LIN {X 0,Y 475.788,Z 378.361,A -85,B 0,C 180,E1 -7451.438,E2 -7451.438} C_VEL
LIN {X 0,Y 475.279,Z 381.668,A -85,B 0,C 180,E1 -7452.005,E2 -7452.005} C_VEL
LIN {X 0,Y 474.286,Z 385.768,A -85,B 0,C 180,E1 -7452.486,E2 -7452.486} C_VEL
LIN {X 0,Y 473.126,Z 390.462,A -85,B 0,C 180,E1 -7452.878,E2 -7452.878} C_VEL
LIN {X 0,Y 471.802,Z 397.453,A -85,B 0,C 180,E1 -7453.254,E2 -7453.254} C_VEL
LIN {X 0,Y 471.382,Z 403.104,A -85,B 0,C 180,E1 -7453.407,E2 -7453.407} C_VEL
LIN {X 0,Y 470.706,Z 494.322,A -85,B 0,C 180,E1 -7454.826,E2 -7454.826} C_VEL
LIN {X 0,Y 470.353,Z 508.19,A -85,B 0,C 180,E1 -7455.23,E2 -7455.23} C_VEL
LIN {X 0,Y 470.018,Z 520.592,A -85,B 0,C 180,E1 -7455.772,E2 -7455.772} C_VEL
LIN {X 0,Y 469.61,Z 532.37,A -85,B 0,C 180,E1 -7456.472,E2 -7456.472} C_VEL
LIN {X 0,Y 469.141,Z 543.794,A -85,B 0,C 180,E1 -7457.345,E2 -7457.345} C_VEL
LIN {X 0,Y 468.592,Z 554.026,A -85,B 0,C 180,E1 -7458.319,E2 -7458.319} C_VEL
LIN {X 0,Y 468.161,Z 563.202,A -85,B 0,C 180,E1 -7459.403,E2 -7459.403} C_VEL
LIN {X 0,Y 467.689,Z 572.108,A -85,B 0,C 180,E1 -7460.704,E2 -7460.704} C_VEL
LIN {X 0,Y 467.314,Z 579.277,A -85,B 0,C 180,E1 -7462.004,E2 -7462.004} C_VEL
LIN {X 0,Y 467.081,Z 584.816,A -85,B 0,C 180,E1 -7463.257,E2 -7463.257} C_VEL
LIN {X 0,Y 466.93,Z 588.808,A -85,B 0,C 180,E1 -7464.386,E2 -7464.386} C_VEL
LIN {X 0,Y 466.822,Z 592.404,A -85,B 0,C 180,E1 -7465.683,E2 -7465.683} C_VEL
LIN {X 0,Y 466.78,Z 594.262,A -85,B 0,C 180,E1 -7466.547,E2 -7466.547} C_VEL
LIN {X 0,Y 466.704,Z 595.664,A -85,B 0,C 180,E1 -7467.411,E2 -7467.411} C_VEL
LIN {X 0,Y 466.62,Z 597.275,A -85,B 0,C 180,E1 -7469.137,E2 -7469.137} C_VEL
LIN {X 0,Y 466.6,Z 597.511,A -85,B 0,C 180,E1 -7470,E2 -7470} C_VEL
LIN {X 0,Y 466.62,Z 597.325,A -85,B 0,C 180,E1 -7470.863,E2 -7470.863} C_VEL
LIN {X 0,Y 466.704,Z 595.778,A -85,B 0,C 180,E1 -7472.589,E2 -7472.589} C_VEL
LIN {X 0,Y 466.78,Z 594.425,A -85,B 0,C 180,E1 -7473.453,E2 -7473.453} C_VEL
LIN {X 0,Y 466.788,Z 591.571,A -85,B 0,C 180,E1 -7474.75,E2 -7474.75} C_VEL
LIN {X 0,Y 467.034,Z 587.692,A -85,B 0,C 180,E1 -7476.046,E2 -7476.046} C_VEL
LIN {X 0,Y 467.17,Z 582.693,A -85,B 0,C 180,E1 -7477.346,E2 -7477.346} C_VEL
LIN {X 0,Y 467.441,Z 576.398,A -85,B 0,C 180,E1 -7478.647,E2 -7478.647} C_VEL
LIN {X 0,Y 467.856,Z 568.513,A -85,B 0,C 180,E1 -7479.947,E2 -7479.947} C_VEL
LIN {X 0,Y 468.293,Z 558.704,A -85,B 0,C 180,E1 -7481.25,E2 -7481.25} C_VEL
LIN {X 0,Y 468.93,Z 548.404,A -85,B 0,C 180,E1 -7482.331,E2 -7482.331} C_VEL
LIN {X 0,Y 469.328,Z 537.488,A -85,B 0,C 180,E1 -7483.256,E2 -7483.256} C_VEL
LIN {X 0,Y 469.796,Z 527.044,A -85,B 0,C 180,E1 -7483.959,E2 -7483.959} C_VEL
LIN {X 0,Y 470.212,Z 514.491,A -85,B 0,C 180,E1 -7484.609,E2 -7484.609} C_VEL
LIN {X 0,Y 470.562,Z 501.002,A -85,B 0,C 180,E1 -7485.095,E2 -7485.095} C_VEL
LIN {X 0,Y 470.722,Z 487.471,A -85,B 0,C 180,E1 -7485.395,E2 -7485.395} C_VEL
LIN {X 0,Y 471.408,Z 402.034,A -85,B 0,C 180,E1 -7486.7,E2 -7486.7} C_VEL
LIN {X 0,Y 468.486,Z 387.239,A -85,B 0,C 180,E1 -7487.057,E2 -7487.057} C_VEL
LIN {X 0,Y 468.974,Z 376.155,A -85,B 0,C 180,E1 -7489.477,E2 -7489.477} C_VEL
LIN {X 0,Y 467.573,Z 368.247,A -85,B 0,C 180,E1 -7491.388,E2 -7491.388} C_VEL
LIN {X 0,Y 467.575,Z 368.247,A -85,B 0,C 180,E1 -7493.943,E2 -7493.943} C_VEL
LIN {X 0,Y 467.617,Z 368.232,A -85,B 0,C 180,E1 -7496.8,E2 -7496.8} C_VEL
LIN {X 0,Y 467.554,Z 368.245,A -85,B 0,C 180,E1 -7499.737,E2 -7499.737} C_VEL
LIN {X 0,Y 467.583,Z 368.236,A -85,B 0,C 180,E1 -7502.758,E2 -7502.758} C_VEL
LIN {X 0,Y 467.555,Z 368.248,A -85,B 0,C 180,E1 -7505.888,E2 -7505.888} C_VEL
LIN {X 0,Y 467.58,Z 368.237,A -85,B 0,C 180,E1 -7509.144,E2 -7509.144} C_VEL
LIN {X 0,Y 467.583,Z 368.236,A -85,B 0,C 180,E1 -7512.566,E2 -7512.566} C_VEL
LIN {X 0,Y 467.567,Z 368.239,A -85,B 0,C 180,E1 -7515.052,E2 -7515.052} C_VEL
LIN {X 0,Y 467.62,Z 368.236,A -85,B 0,C 180,E1 -7517.443,E2 -7517.443} C_VEL
LIN {X 0,Y 467.595,Z 368.235,A -85,B 0,C 180,E1 -7520.856,E2 -7520.856} C_VEL
LIN {X 0,Y 467.558,Z 368.24,A -85,B 0,C 180,E1 -7524.26,E2 -7524.26} C_VEL
LIN {X 0,Y 467.583,Z 368.241,A -85,B 0,C 180,E1 -7527.319,E2 -7527.319} C_VEL
LIN {X 0,Y 467.563,Z 368.239,A -85,B 0,C 180,E1 -7530.667,E2 -7530.667} C_VEL
LIN {X 0,Y 467.621,Z 368.236,A -85,B 0,C 180,E1 -7533.2,E2 -7533.2} C_VEL
LIN {X 0,Y 467.586,Z 368.236,A -85,B 0,C 180,E1 -7536.467,E2 -7536.467} C_VEL
LIN {X 0,Y 467.616,Z 368.235,A -85,B 0,C 180,E1 -7539.777,E2 -7539.777} C_VEL
LIN {X 0,Y 467.601,Z 368.234,A -85,B 0,C 180,E1 -7542.506,E2 -7542.506} C_VEL
LIN {X 0,Y 467.601,Z 368.241,A -85,B 0,C 180,E1 -7545.196,E2 -7545.196} C_VEL
LIN {X 0,Y 467.674,Z 368.226,A -85,B 0,C 180,E1 -7547.855,E2 -7547.855} C_VEL
LIN {X 0,Y 467.674,Z 368.231,A -85,B 0,C 180,E1 -7551.357,E2 -7551.357} C_VEL
LIN {X 0,Y 467.735,Z 368.218,A -85,B 0,C 180,E1 -7553.962,E2 -7553.962} C_VEL
LIN {X 0,Y 467.853,Z 368.207,A -85,B 0,C 180,E1 -7557.417,E2 -7557.417} C_VEL
LIN {X 0,Y 467.873,Z 368.2,A -85,B 0,C 180,E1 -7560,E2 -7560} C_VEL
LIN {X 0,Y 467.853,Z 368.205,A -85,B 0,C 180,E1 -7562.583,E2 -7562.583} C_VEL
LIN {X 0,Y 467.739,Z 368.217,A -85,B 0,C 180,E1 -7566.037,E2 -7566.037} C_VEL
LIN {X 0,Y 467.674,Z 368.228,A -85,B 0,C 180,E1 -7568.643,E2 -7568.643} C_VEL
LIN {X 0,Y 467.674,Z 368.225,A -85,B 0,C 180,E1 -7572.145,E2 -7572.145} C_VEL
LIN {X 0,Y 467.641,Z 368.229,A -85,B 0,C 180,E1 -7575.886,E2 -7575.886} C_VEL
LIN {X 0,Y 467.616,Z 368.234,A -85,B 0,C 180,E1 -7579.308,E2 -7579.308} C_VEL
LIN {X 0,Y 467.534,Z 368.243,A -85,B 0,C 180,E1 -7582.074,E2 -7582.074} C_VEL
LIN {X 0,Y 467.598,Z 368.241,A -85,B 0,C 180,E1 -7584.888,E2 -7584.888} C_VEL
LIN {X 0,Y 467.62,Z 368.232,A -85,B 0,C 180,E1 -7587.769,E2 -7587.769} C_VEL
LIN {X 0,Y 467.562,Z 368.242,A -85,B 0,C 180,E1 -7591.046,E2 -7591.046} C_VEL
LIN {X 0,Y 467.584,Z 368.239,A -85,B 0,C 180,E1 -7594.243,E2 -7594.243} C_VEL
LIN {X 0,Y 467.545,Z 368.242,A -85,B 0,C 180,E1 -7597.188,E2 -7597.188} C_VEL
LIN {X 0,Y 467.591,Z 368.24,A -85,B 0,C 180,E1 -7600.263,E2 -7600.263} C_VEL
LIN {X 0,Y 467.615,Z 368.24,A -85,B 0,C 180,E1 -7602.572,E2 -7602.572} C_VEL
LIN {X 0,Y 467.563,Z 368.243,A -85,B 0,C 180,E1 -7606.178,E2 -7606.178} C_VEL
LIN {X 0,Y 467.579,Z 368.241,A -85,B 0,C 180,E1 -7608.723,E2 -7608.723} C_VEL
LIN {X 0,Y 467.564,Z 368.242,A -85,B 0,C 180,E1 -7611.956,E2 -7611.956} C_VEL
LIN {X 0,Y 467.567,Z 368.238,A -85,B 0,C 180,E1 -7615.169,E2 -7615.169} C_VEL
LIN {X 0,Y 467.583,Z 368.244,A -85,B 0,C 180,E1 -7618.261,E2 -7618.261} C_VEL
LIN {X 0,Y 467.576,Z 368.241,A -85,B 0,C 180,E1 -7621.251,E2 -7621.251} C_VEL
LIN {X 0,Y 467.669,Z 368.367,A -85,B 0,C 180,E1 -7623.805,E2 -7623.805} C_VEL
LIN {X 0,Y 469.783,Z 379.089,A -85,B 0,C 180,E1 -7625.863,E2 -7625.863} C_VEL
LIN {X 0,Y 469.854,Z 384.768,A -85,B 0,C 180,E1 -7626.882,E2 -7626.882} C_VEL
LIN {X 0,Y 469.109,Z 400.416,A -85,B 0,C 180,E1 -7629.616,E2 -7629.616} C_VEL
LIN {X 0,Y 468.442,Z 417.254,A -85,B 0,C 180,E1 -7632.539,E2 -7632.539} C_VEL
LIN {X 0,Y 468.328,Z 419.783,A -85,B 0,C 180,E1 -7632.978,E2 -7632.978} C_VEL
LIN {X 0,Y 471.197,Z 439.463,A -85,B 0,C 180,E1 -7633.391,E2 -7633.391} C_VEL
LIN {X 0,Y 470.547,Z 528.128,A -85,B 0,C 180,E1 -7634.765,E2 -7634.765} C_VEL
LIN {X 0,Y 470.162,Z 541.402,A -85,B 0,C 180,E1 -7635.141,E2 -7635.141} C_VEL
LIN {X 0,Y 469.689,Z 554.694,A -85,B 0,C 180,E1 -7635.707,E2 -7635.707} C_VEL
LIN {X 0,Y 469.247,Z 565.855,A -85,B 0,C 180,E1 -7636.356,E2 -7636.356} C_VEL
LIN {X 0,Y 468.69,Z 577.047,A -85,B 0,C 180,E1 -7637.187,E2 -7637.187} C_VEL
LIN {X 0,Y 468.235,Z 587.923,A -85,B 0,C 180,E1 -7638.2,E2 -7638.2} C_VEL
LIN {X 0,Y 467.784,Z 596.474,A -85,B 0,C 180,E1 -7639.176,E2 -7639.176} C_VEL
LIN {X 0,Y 467.434,Z 604.368,A -85,B 0,C 180,E1 -7640.262,E2 -7640.262} C_VEL
LIN {X 0,Y 467.113,Z 612.079,A -85,B 0,C 180,E1 -7641.565,E2 -7641.565} C_VEL
LIN {X 0,Y 466.858,Z 619.19,A -85,B 0,C 180,E1 -7643.083,E2 -7643.083} C_VEL
LIN {X 0,Y 466.763,Z 623.924,A -85,B 0,C 180,E1 -7644.384,E2 -7644.384} C_VEL
LIN {X 0,Y 466.648,Z 627.539,A -85,B 0,C 180,E1 -7645.681,E2 -7645.681} C_VEL
LIN {X 0,Y 466.69,Z 629.407,A -85,B 0,C 180,E1 -7646.547,E2 -7646.547} C_VEL
LIN {X 0,Y 466.662,Z 630.806,A -85,B 0,C 180,E1 -7647.411,E2 -7647.411} C_VEL
LIN {X 0,Y 466.619,Z 632.413,A -85,B 0,C 180,E1 -7649.137,E2 -7649.137} C_VEL
LIN {X 0,Y 466.599,Z 632.629,A -85,B 0,C 180,E1 -7650,E2 -7650} C_VEL
LIN {X 0,Y 466.619,Z 632.413,A -85,B 0,C 180,E1 -7650.863,E2 -7650.863} C_VEL
LIN {X 0,Y 466.662,Z 630.809,A -85,B 0,C 180,E1 -7652.589,E2 -7652.589} C_VEL
LIN {X 0,Y 466.69,Z 629.41,A -85,B 0,C 180,E1 -7653.453,E2 -7653.453} C_VEL
LIN {X 0,Y 466.69,Z 626.466,A -85,B 0,C 180,E1 -7654.751,E2 -7654.751} C_VEL
LIN {X 0,Y 466.753,Z 622.483,A -85,B 0,C 180,E1 -7656.05,E2 -7656.05} C_VEL
LIN {X 0,Y 466.943,Z 616.362,A -85,B 0,C 180,E1 -7657.567,E2 -7657.567} C_VEL
LIN {X 0,Y 467.188,Z 609.672,A -85,B 0,C 180,E1 -7658.87,E2 -7658.87} C_VEL
LIN {X 0,Y 467.521,Z 601.374,A -85,B 0,C 180,E1 -7660.173,E2 -7660.173} C_VEL
LIN {X 0,Y 468.007,Z 592.876,A -85,B 0,C 180,E1 -7661.257,E2 -7661.257} C_VEL
LIN {X 0,Y 468.474,Z 582.834,A -85,B 0,C 180,E1 -7662.301,E2 -7662.301} C_VEL
LIN {X 0,Y 468.938,Z 571.987,A -85,B 0,C 180,E1 -7663.212,E2 -7663.212} C_VEL
LIN {X 0,Y 469.449,Z 560.604,A -85,B 0,C 180,E1 -7663.969,E2 -7663.969} C_VEL
LIN {X 0,Y 469.913,Z 548.932,A -85,B 0,C 180,E1 -7664.563,E2 -7664.563} C_VEL
LIN {X 0,Y 470.33,Z 536.401,A -85,B 0,C 180,E1 -7665.02,E2 -7665.02} C_VEL
LIN {X 0,Y 470.645,Z 523.722,A -85,B 0,C 180,E1 -7665.314,E2 -7665.314} C_VEL
LIN {X 0,Y 471.1,Z 437.824,A -85,B 0,C 180,E1 -7666.636,E2 -7666.636} C_VEL
LIN {X 0,Y 468.331,Z 419.732,A -85,B 0,C 180,E1 -7667.032,E2 -7667.032} C_VEL
LIN {X 0,Y 469.063,Z 401.69,A -85,B 0,C 180,E1 -7670.158,E2 -7670.158} C_VEL
LIN {X 0,Y 469.826,Z 386.056,A -85,B 0,C 180,E1 -7672.887,E2 -7672.887} C_VEL
LIN {X 0,Y 469.981,Z 380.833,A -85,B 0,C 180,E1 -7673.812,E2 -7673.812} C_VEL
LIN {X 0,Y 468.071,Z 370.311,A -85,B 0,C 180,E1 -7675.812,E2 -7675.812} C_VEL
LIN {X 0,Y 467.645,Z 368.234,A -85,B 0,C 180,E1 -7676.257,E2 -7676.257} C_VEL
LIN {X 0,Y 467.57,Z 368.244,A -85,B 0,C 180,E1 -7679.332,E2 -7679.332} C_VEL
LIN {X 0,Y 467.581,Z 368.236,A -85,B 0,C 180,E1 -7682.679,E2 -7682.679} C_VEL
LIN {X 0,Y 467.561,Z 368.246,A -85,B 0,C 180,E1 -7685.739,E2 -7685.739} C_VEL
LIN {X 0,Y 467.58,Z 368.239,A -85,B 0,C 180,E1 -7689.144,E2 -7689.144} C_VEL
LIN {X 0,Y 467.583,Z 368.236,A -85,B 0,C 180,E1 -7692.566,E2 -7692.566} C_VEL
LIN {X 0,Y 467.567,Z 368.24,A -85,B 0,C 180,E1 -7695.052,E2 -7695.052} C_VEL
LIN {X 0,Y 467.62,Z 368.239,A -85,B 0,C 180,E1 -7697.443,E2 -7697.443} C_VEL
LIN {X 0,Y 467.61,Z 368.234,A -85,B 0,C 180,E1 -7700.858,E2 -7700.858} C_VEL
LIN {X 0,Y 467.557,Z 368.24,A -85,B 0,C 180,E1 -7704.26,E2 -7704.26} C_VEL
LIN {X 0,Y 467.576,Z 368.245,A -85,B 0,C 180,E1 -7707.32,E2 -7707.32} C_VEL
LIN {X 0,Y 467.571,Z 368.238,A -85,B 0,C 180,E1 -7710.665,E2 -7710.665} C_VEL
LIN {X 0,Y 467.621,Z 368.238,A -85,B 0,C 180,E1 -7713.2,E2 -7713.2} C_VEL
LIN {X 0,Y 467.586,Z 368.236,A -85,B 0,C 180,E1 -7716.467,E2 -7716.467} C_VEL
LIN {X 0,Y 467.616,Z 368.234,A -85,B 0,C 180,E1 -7719.777,E2 -7719.777} C_VEL
LIN {X 0,Y 467.601,Z 368.235,A -85,B 0,C 180,E1 -7722.506,E2 -7722.506} C_VEL
LIN {X 0,Y 467.599,Z 368.242,A -85,B 0,C 180,E1 -7725.196,E2 -7725.196} C_VEL
LIN {X 0,Y 467.674,Z 368.225,A -85,B 0,C 180,E1 -7727.855,E2 -7727.855} C_VEL
LIN {X 0,Y 467.674,Z 368.229,A -85,B 0,C 180,E1 -7731.357,E2 -7731.357} C_VEL
LIN {X 0,Y 467.735,Z 368.217,A -85,B 0,C 180,E1 -7733.963,E2 -7733.963} C_VEL
LIN {X 0,Y 467.853,Z 368.205,A -85,B 0,C 180,E1 -7737.417,E2 -7737.417} C_VEL
LIN {X 0,Y 467.873,Z 368.2,A -85,B 0,C 180,E1 -7740,E2 -7740} C_VEL
LIN {X 0,Y 467.853,Z 368.206,A -85,B 0,C 180,E1 -7742.583,E2 -7742.583} C_VEL
LIN {X 0,Y 467.739,Z 368.217,A -85,B 0,C 180,E1 -7746.038,E2 -7746.038} C_VEL
LIN {X 0,Y 467.674,Z 368.231,A -85,B 0,C 180,E1 -7748.643,E2 -7748.643} C_VEL
LIN {X 0,Y 467.674,Z 368.226,A -85,B 0,C 180,E1 -7752.145,E2 -7752.145} C_VEL
LIN {X 0,Y 467.641,Z 368.229,A -85,B 0,C 180,E1 -7755.886,E2 -7755.886} C_VEL
LIN {X 0,Y 467.616,Z 368.233,A -85,B 0,C 180,E1 -7759.308,E2 -7759.308} C_VEL
LIN {X 0,Y 467.535,Z 368.244,A -85,B 0,C 180,E1 -7762.074,E2 -7762.074} C_VEL
LIN {X 0,Y 467.598,Z 368.239,A -85,B 0,C 180,E1 -7764.888,E2 -7764.888} C_VEL
LIN {X 0,Y 467.62,Z 368.232,A -85,B 0,C 180,E1 -7767.769,E2 -7767.769} C_VEL
LIN {X 0,Y 467.562,Z 368.241,A -85,B 0,C 180,E1 -7771.046,E2 -7771.046} C_VEL
LIN {X 0,Y 467.584,Z 368.241,A -85,B 0,C 180,E1 -7774.243,E2 -7774.243} C_VEL
LIN {X 0,Y 467.545,Z 368.241,A -85,B 0,C 180,E1 -7777.187,E2 -7777.187} C_VEL
LIN {X 0,Y 467.592,Z 368.242,A -85,B 0,C 180,E1 -7780.263,E2 -7780.263} C_VEL
LIN {X 0,Y 467.615,Z 368.237,A -85,B 0,C 180,E1 -7782.572,E2 -7782.572} C_VEL
LIN {X 0,Y 467.567,Z 368.239,A -85,B 0,C 180,E1 -7785.054,E2 -7785.054} C_VEL
LIN {X 0,Y 467.586,Z 368.236,A -85,B 0,C 180,E1 -7787.441,E2 -7787.441} C_VEL
LIN {X 0,Y 467.58,Z 368.238,A -85,B 0,C 180,E1 -7790.856,E2 -7790.856} C_VEL
LIN {X 0,Y 467.562,Z 368.246,A -85,B 0,C 180,E1 -7794.261,E2 -7794.261} C_VEL
LIN {X 0,Y 467.581,Z 368.237,A -85,B 0,C 180,E1 -7797.322,E2 -7797.322} C_VEL
LIN {X 0,Y 467.571,Z 368.239,A -85,B 0,C 180,E1 -7800.668,E2 -7800.668} C_VEL
LIN {X 0,Y 467.613,Z 368.232,A -85,B 0,C 180,E1 -7803.2,E2 -7803.2} C_VEL
LIN {X 0,Y 467.592,Z 368.242,A -85,B 0,C 180,E1 -7806.469,E2 -7806.469} C_VEL
LIN {X 0,Y 467.613,Z 368.349,A -85,B 0,C 180,E1 -7808.782,E2 -7808.782} C_VEL
LIN {X 0,Y 468.894,Z 375.745,A -85,B 0,C 180,E1 -7810.52,E2 -7810.52} C_VEL
LIN {X 0,Y 468.522,Z 387.257,A -85,B 0,C 180,E1 -7813.042,E2 -7813.042} C_VEL
LIN {X 0,Y 471.391,Z 401.608,A -85,B 0,C 180,E1 -7813.384,E2 -7813.384} C_VEL
LIN {X 0,Y 471.382,Z 403.104,A -85,B 0,C 180,E1 -7813.407,E2 -7813.407} C_VEL
LIN {X 0,Y 470.725,Z 408.947,A -85,B 0,C 180,E1 -7813.474,E2 -7813.474} C_VEL
LIN {X 0,Y 465.159,Z 427.969,A -85,B 0,C 180,E1 -7813.568,E2 -7813.568} C_VEL
LIN {X 0,Y 464.425,Z 433.815,A -85,B 0,C 180,E1 -7813.633,E2 -7813.633} C_VEL
LIN {X 0,Y 463.89,Z 494.607,A -85,B 0,C 180,E1 -7814.598,E2 -7814.598} C_VEL
LIN {X 0,Y 463.509,Z 508.469,A -85,B 0,C 180,E1 -7815.007,E2 -7815.007} C_VEL
LIN {X 0,Y 463.16,Z 520.867,A -85,B 0,C 180,E1 -7815.557,E2 -7815.557} C_VEL
LIN {X 0,Y 462.766,Z 531.297,A -85,B 0,C 180,E1 -7816.173,E2 -7816.173} C_VEL
LIN {X 0,Y 462.268,Z 542.781,A -85,B 0,C 180,E1 -7817.042,E2 -7817.042} C_VEL
LIN {X 0,Y 461.669,Z 553.239,A -85,B 0,C 180,E1 -7818.029,E2 -7818.029} C_VEL
LIN {X 0,Y 461.265,Z 561.778,A -85,B 0,C 180,E1 -7819.021,E2 -7819.021} C_VEL
LIN {X 0,Y 460.804,Z 569.644,A -85,B 0,C 180,E1 -7820.121,E2 -7820.121} C_VEL
LIN {X 0,Y 460.394,Z 577.331,A -85,B 0,C 180,E1 -7821.441,E2 -7821.441} C_VEL
LIN {X 0,Y 460.053,Z 584.381,A -85,B 0,C 180,E1 -7822.98,E2 -7822.98} C_VEL
LIN {X 0,Y 459.886,Z 589.076,A -85,B 0,C 180,E1 -7824.299,E2 -7824.299} C_VEL
LIN {X 0,Y 459.729,Z 592.673,A -85,B 0,C 180,E1 -7825.616,E2 -7825.616} C_VEL
LIN {X 0,Y 459.716,Z 594.529,A -85,B 0,C 180,E1 -7826.494,E2 -7826.494} C_VEL
LIN {X 0,Y 459.626,Z 595.932,A -85,B 0,C 180,E1 -7827.371,E2 -7827.371} C_VEL
LIN {X 0,Y 459.553,Z 597.542,A -85,B 0,C 180,E1 -7829.124,E2 -7829.124} C_VEL
LIN {X 0,Y 459.532,Z 597.777,A -85,B 0,C 180,E1 -7830,E2 -7830} C_VEL
LIN {X 0,Y 459.553,Z 597.591,A -85,B 0,C 180,E1 -7830.876,E2 -7830.876} C_VEL
LIN {X 0,Y 459.626,Z 596.044,A -85,B 0,C 180,E1 -7832.629,E2 -7832.629} C_VEL
LIN {X 0,Y 459.716,Z 594.691,A -85,B 0,C 180,E1 -7833.506,E2 -7833.506} C_VEL
LIN {X 0,Y 459.706,Z 591.837,A -85,B 0,C 180,E1 -7834.823,E2 -7834.823} C_VEL
LIN {X 0,Y 459.982,Z 587.957,A -85,B 0,C 180,E1 -7836.139,E2 -7836.139} C_VEL
LIN {X 0,Y 460.125,Z 582.958,A -85,B 0,C 180,E1 -7837.46,E2 -7837.46} C_VEL
LIN {X 0,Y 460.412,Z 576.664,A -85,B 0,C 180,E1 -7838.78,E2 -7838.78} C_VEL
LIN {X 0,Y 460.849,Z 568.778,A -85,B 0,C 180,E1 -7840.1,E2 -7840.1} C_VEL
LIN {X 0,Y 461.349,Z 558.967,A -85,B 0,C 180,E1 -7841.422,E2 -7841.422} C_VEL
LIN {X 0,Y 462.004,Z 548.666,A -85,B 0,C 180,E1 -7842.519,E2 -7842.519} C_VEL
LIN {X 0,Y 462.458,Z 537.174,A -85,B 0,C 180,E1 -7843.502,E2 -7843.502} C_VEL
LIN {X 0,Y 463.001,Z 525.482,A -85,B 0,C 180,E1 -7844.28,E2 -7844.28} C_VEL
LIN {X 0,Y 463.455,Z 513.448,A -85,B 0,C 180,E1 -7844.883,E2 -7844.883} C_VEL
LIN {X 0,Y 463.787,Z 500.338,A -85,B 0,C 180,E1 -7845.35,E2 -7845.35} C_VEL
LIN {X 0,Y 463.899,Z 487.708,A -85,B 0,C 180,E1 -7845.627,E2 -7845.627} C_VEL
LIN {X 0,Y 464.614,Z 403.405,A -85,B 0,C 180,E1 -7846.933,E2 -7846.933} C_VEL
LIN {X 0,Y 461.574,Z 387.453,A -85,B 0,C 180,E1 -7847.329,E2 -7847.329} C_VEL
LIN {X 0,Y 461.94,Z 376.384,A -85,B 0,C 180,E1 -7849.786,E2 -7849.786} C_VEL
LIN {X 0,Y 460.521,Z 369.126,A -85,B 0,C 180,E1 -7851.544,E2 -7851.544} C_VEL
LIN {X 0,Y 460.544,Z 369.123,A -85,B 0,C 180,E1 -7854.332,E2 -7854.332} C_VEL
LIN {X 0,Y 460.573,Z 369.11,A -85,B 0,C 180,E1 -7857.243,E2 -7857.243} C_VEL
LIN {X 0,Y 460.51,Z 369.122,A -85,B 0,C 180,E1 -7860.239,E2 -7860.239} C_VEL
LIN {X 0,Y 460.529,Z 369.116,A -85,B 0,C 180,E1 -7863.324,E2 -7863.324} C_VEL
LIN {X 0,Y 460.478,Z 369.122,A -85,B 0,C 180,E1 -7866.528,E2 -7866.528} C_VEL
LIN {X 0,Y 460.555,Z 369.119,A -85,B 0,C 180,E1 -7869.859,E2 -7869.859} C_VEL
LIN {X 0,Y 460.51,Z 369.117,A -85,B 0,C 180,E1 -7872.9,E2 -7872.9} C_VEL
LIN {X 0,Y 460.52,Z 369.123,A -85,B 0,C 180,E1 -7875.828,E2 -7875.828} C_VEL
LIN {X 0,Y 460.539,Z 369.114,A -85,B 0,C 180,E1 -7878.989,E2 -7878.989} C_VEL
LIN {X 0,Y 460.534,Z 369.117,A -85,B 0,C 180,E1 -7881.268,E2 -7881.268} C_VEL
LIN {X 0,Y 460.508,Z 369.117,A -85,B 0,C 180,E1 -7884.554,E2 -7884.554} C_VEL
LIN {X 0,Y 460.53,Z 369.121,A -85,B 0,C 180,E1 -7887.715,E2 -7887.715} C_VEL
LIN {X 0,Y 460.533,Z 369.115,A -85,B 0,C 180,E1 -7890.768,E2 -7890.768} C_VEL
LIN {X 0,Y 460.561,Z 369.116,A -85,B 0,C 180,E1 -7893.734,E2 -7893.734} C_VEL
LIN {X 0,Y 460.54,Z 369.114,A -85,B 0,C 180,E1 -7896.624,E2 -7896.624} C_VEL
LIN {X 0,Y 460.546,Z 369.12,A -85,B 0,C 180,E1 -7899.452,E2 -7899.452} C_VEL
LIN {X 0,Y 460.551,Z 369.112,A -85,B 0,C 180,E1 -7902.23,E2 -7902.23} C_VEL
LIN {X 0,Y 460.559,Z 369.115,A -85,B 0,C 180,E1 -7904.965,E2 -7904.965} C_VEL
LIN {X 0,Y 460.621,Z 369.107,A -85,B 0,C 180,E1 -7907.666,E2 -7907.666} C_VEL
LIN {X 0,Y 460.621,Z 369.112,A -85,B 0,C 180,E1 -7911.224,E2 -7911.224} C_VEL
LIN {X 0,Y 460.701,Z 369.094,A -85,B 0,C 180,E1 -7913.87,E2 -7913.87} C_VEL
LIN {X 0,Y 460.818,Z 369.084,A -85,B 0,C 180,E1 -7917.378,E2 -7917.378} C_VEL
LIN {X 0,Y 460.844,Z 369.076,A -85,B 0,C 180,E1 -7920,E2 -7920} C_VEL
LIN {X 0,Y 460.818,Z 369.081,A -85,B 0,C 180,E1 -7922.622,E2 -7922.622} C_VEL
LIN {X 0,Y 460.704,Z 369.093,A -85,B 0,C 180,E1 -7926.13,E2 -7926.13} C_VEL
LIN {X 0,Y 460.622,Z 369.109,A -85,B 0,C 180,E1 -7928.776,E2 -7928.776} C_VEL
LIN {X 0,Y 460.625,Z 369.105,A -85,B 0,C 180,E1 -7932.457,E2 -7932.457} C_VEL
LIN {X 0,Y 460.591,Z 369.107,A -85,B 0,C 180,E1 -7935.998,E2 -7935.998} C_VEL
LIN {X 0,Y 460.563,Z 369.118,A -85,B 0,C 180,E1 -7938.902,E2 -7938.902} C_VEL
LIN {X 0,Y 460.511,Z 369.118,A -85,B 0,C 180,E1 -7941.486,E2 -7941.486} C_VEL
LIN {X 0,Y 460.537,Z 369.117,A -85,B 0,C 180,E1 -7944.333,E2 -7944.333} C_VEL
LIN {X 0,Y 460.577,Z 369.111,A -85,B 0,C 180,E1 -7947.244,E2 -7947.244} C_VEL
LIN {X 0,Y 460.504,Z 369.121,A -85,B 0,C 180,E1 -7950.241,E2 -7950.241} C_VEL
LIN {X 0,Y 460.523,Z 369.116,A -85,B 0,C 180,E1 -7953.325,E2 -7953.325} C_VEL
LIN {X 0,Y 460.473,Z 369.129,A -85,B 0,C 180,E1 -7956.53,E2 -7956.53} C_VEL
LIN {X 0,Y 460.571,Z 369.111,A -85,B 0,C 180,E1 -7959.858,E2 -7959.858} C_VEL
LIN {X 0,Y 460.538,Z 369.117,A -85,B 0,C 180,E1 -7962.905,E2 -7962.905} C_VEL
LIN {X 0,Y 460.515,Z 369.118,A -85,B 0,C 180,E1 -7965.83,E2 -7965.83} C_VEL
LIN {X 0,Y 460.531,Z 369.116,A -85,B 0,C 180,E1 -7968.99,E2 -7968.99} C_VEL
LIN {X 0,Y 460.524,Z 369.116,A -85,B 0,C 180,E1 -7971.268,E2 -7971.268} C_VEL
LIN {X 0,Y 460.512,Z 369.122,A -85,B 0,C 180,E1 -7974.555,E2 -7974.555} C_VEL
LIN {X 0,Y 460.531,Z 369.116,A -85,B 0,C 180,E1 -7977.716,E2 -7977.716} C_VEL
LIN {X 0,Y 460.539,Z 369.118,A -85,B 0,C 180,E1 -7980.77,E2 -7980.77} C_VEL
LIN {X 0,Y 460.608,Z 369.277,A -85,B 0,C 180,E1 -7983.586,E2 -7983.586} C_VEL
LIN {X 0,Y 462.885,Z 380.608,A -85,B 0,C 180,E1 -7985.799,E2 -7985.799} C_VEL
LIN {X 0,Y 462.909,Z 387.144,A -85,B 0,C 180,E1 -7986.987,E2 -7986.987} C_VEL
LIN {X 0,Y 461.889,Z 406.654,A -85,B 0,C 180,E1 -7990.443,E2 -7990.443} C_VEL
LIN {X 0,Y 461.353,Z 419.521,A -85,B 0,C 180,E1 -7992.712,E2 -7992.712} C_VEL
LIN {X 0,Y 464.387,Z 439.503,A -85,B 0,C 180,E1 -7993.145,E2 -7993.145} C_VEL
LIN {X 0,Y 463.698,Z 527.871,A -85,B 0,C 180,E1 -7994.535,E2 -7994.535} C_VEL
LIN {X 0,Y 463.317,Z 541.142,A -85,B 0,C 180,E1 -7994.916,E2 -7994.916} C_VEL
LIN {X 0,Y 462.795,Z 554.431,A -85,B 0,C 180,E1 -7995.489,E2 -7995.489} C_VEL
LIN {X 0,Y 462.324,Z 565.59,A -85,B 0,C 180,E1 -7996.148,E2 -7996.148} C_VEL
LIN {X 0,Y 461.705,Z 577.661,A -85,B 0,C 180,E1 -7997.065,E2 -7997.065} C_VEL
LIN {X 0,Y 461.207,Z 588.703,A -85,B 0,C 180,E1 -7998.129,E2 -7998.129} C_VEL
LIN {X 0,Y 460.685,Z 597.889,A -85,B 0,C 180,E1 -7999.229,E2 -7999.229} C_VEL
LIN {X 0,Y 460.266,Z 606.845,A -85,B 0,C 180,E1 -8000.553,E2 -8000.553} C_VEL
LIN {X 0,Y 459.954,Z 614.055,A -85,B 0,C 180,E1 -8001.875,E2 -8001.875} C_VEL
LIN {X 0,Y 459.776,Z 618.923,A -85,B 0,C 180,E1 -8002.976,E2 -8002.976} C_VEL
LIN {X 0,Y 459.659,Z 623.656,A -85,B 0,C 180,E1 -8004.297,E2 -8004.297} C_VEL
LIN {X 0,Y 459.565,Z 627.272,A -85,B 0,C 180,E1 -8005.615,E2 -8005.615} C_VEL
LIN {X 0,Y 459.586,Z 629.14,A -85,B 0,C 180,E1 -8006.493,E2 -8006.493} C_VEL
LIN {X 0,Y 459.584,Z 630.54,A -85,B 0,C 180,E1 -8007.371,E2 -8007.371} C_VEL
LIN {X 0,Y 459.552,Z 632.147,A -85,B 0,C 180,E1 -8009.124,E2 -8009.124} C_VEL
LIN {X 0,Y 459.53,Z 632.363,A -85,B 0,C 180,E1 -8010,E2 -8010} C_VEL
LIN {X 0,Y 459.552,Z 632.147,A -85,B 0,C 180,E1 -8010.876,E2 -8010.876} C_VEL
LIN {X 0,Y 459.584,Z 630.542,A -85,B 0,C 180,E1 -8012.629,E2 -8012.629} C_VEL
LIN {X 0,Y 459.586,Z 629.142,A -85,B 0,C 180,E1 -8013.507,E2 -8013.507} C_VEL
LIN {X 0,Y 459.617,Z 626.199,A -85,B 0,C 180,E1 -8014.824,E2 -8014.824} C_VEL
LIN {X 0,Y 459.714,Z 621.183,A -85,B 0,C 180,E1 -8016.431,E2 -8016.431} C_VEL
LIN {X 0,Y 459.894,Z 615.077,A -85,B 0,C 180,E1 -8017.905,E2 -8017.905} C_VEL
LIN {X 0,Y 460.209,Z 608.163,A -85,B 0,C 180,E1 -8019.227,E2 -8019.227} C_VEL
LIN {X 0,Y 460.585,Z 599.515,A -85,B 0,C 180,E1 -8020.55,E2 -8020.55} C_VEL
LIN {X 0,Y 461.098,Z 590.652,A -85,B 0,C 180,E1 -8021.651,E2 -8021.651} C_VEL
LIN {X 0,Y 461.598,Z 579.8,A -85,B 0,C 180,E1 -8022.749,E2 -8022.749} C_VEL
LIN {X 0,Y 462.198,Z 568.744,A -85,B 0,C 180,E1 -8023.632,E2 -8023.632} C_VEL
LIN {X 0,Y 462.706,Z 556.413,A -85,B 0,C 180,E1 -8024.401,E2 -8024.401} C_VEL
LIN {X 0,Y 463.233,Z 543.373,A -85,B 0,C 180,E1 -8025.002,E2 -8025.002} C_VEL
LIN {X 0,Y 463.665,Z 530.079,A -85,B 0,C 180,E1 -8025.41,E2 -8025.41} C_VEL
LIN {X 0,Y 463.936,Z 509.4,A -85,B 0,C 180,E1 -8025.767,E2 -8025.767} C_VEL
LIN {X 0,Y 464.303,Z 438.62,A -85,B 0,C 180,E1 -8026.87,E2 -8026.87} C_VEL
LIN {X 0,Y 461.356,Z 419.522,A -85,B 0,C 180,E1 -8027.287,E2 -8027.287} C_VEL
LIN {X 0,Y 462.088,Z 402.74,A -85,B 0,C 180,E1 -8030.243,E2 -8030.243} C_VEL
LIN {X 0,Y 462.902,Z 387.124,A -85,B 0,C 180,E1 -8033.013,E2 -8033.013} C_VEL
LIN {X 0,Y 462.885,Z 380.592,A -85,B 0,C 180,E1 -8034.201,E2 -8034.201} C_VEL
LIN {X 0,Y 460.588,Z 369.112,A -85,B 0,C 180,E1 -8036.446,E2 -8036.446} C_VEL
LIN {X 0,Y 460.531,Z 369.122,A -85,B 0,C 180,E1 -8039.558,E2 -8039.558} C_VEL
LIN {X 0,Y 460.531,Z 369.119,A -85,B 0,C 180,E1 -8042.284,E2 -8042.284} C_VEL
LIN {X 0,Y 460.512,Z 369.122,A -85,B 0,C 180,E1 -8045.445,E2 -8045.445} C_VEL
LIN {X 0,Y 460.542,Z 369.114,A -85,B 0,C 180,E1 -8048.897,E2 -8048.897} C_VEL
LIN {X 0,Y 460.52,Z 369.117,A -85,B 0,C 180,E1 -8052.18,E2 -8052.18} C_VEL
LIN {X 0,Y 460.518,Z 369.123,A -85,B 0,C 180,E1 -8055.411,E2 -8055.411} C_VEL
LIN {X 0,Y 460.541,Z 369.114,A -85,B 0,C 180,E1 -8058.395,E2 -8058.395} C_VEL
LIN {X 0,Y 460.539,Z 369.119,A -85,B 0,C 180,E1 -8061.268,E2 -8061.268} C_VEL
LIN {X 0,Y 460.508,Z 369.118,A -85,B 0,C 180,E1 -8064.554,E2 -8064.554} C_VEL
LIN {X 0,Y 460.526,Z 369.119,A -85,B 0,C 180,E1 -8067.715,E2 -8067.715} C_VEL
LIN {X 0,Y 460.54,Z 369.115,A -85,B 0,C 180,E1 -8070.769,E2 -8070.769} C_VEL
LIN {X 0,Y 460.561,Z 369.114,A -85,B 0,C 180,E1 -8073.735,E2 -8073.735} C_VEL
LIN {X 0,Y 460.54,Z 369.115,A -85,B 0,C 180,E1 -8076.624,E2 -8076.624} C_VEL
LIN {X 0,Y 460.546,Z 369.118,A -85,B 0,C 180,E1 -8079.452,E2 -8079.452} C_VEL
LIN {X 0,Y 460.551,Z 369.112,A -85,B 0,C 180,E1 -8082.23,E2 -8082.23} C_VEL
LIN {X 0,Y 460.557,Z 369.117,A -85,B 0,C 180,E1 -8084.965,E2 -8084.965} C_VEL
LIN {X 0,Y 460.62,Z 369.105,A -85,B 0,C 180,E1 -8087.666,E2 -8087.666} C_VEL
LIN {X 0,Y 460.621,Z 369.109,A -85,B 0,C 180,E1 -8091.224,E2 -8091.224} C_VEL
LIN {X 0,Y 460.701,Z 369.094,A -85,B 0,C 180,E1 -8093.87,E2 -8093.87} C_VEL
LIN {X 0,Y 460.818,Z 369.082,A -85,B 0,C 180,E1 -8097.378,E2 -8097.378} C_VEL
LIN {X 0,Y 460.844,Z 369.076,A -85,B 0,C 180,E1 -8100,E2 -8100} C_VEL
LIN {X 0,Y 460.818,Z 369.083,A -85,B 0,C 180,E1 -8102.622,E2 -8102.622} C_VEL
LIN {X 0,Y 460.704,Z 369.094,A -85,B 0,C 180,E1 -8106.13,E2 -8106.13} C_VEL
LIN {X 0,Y 460.621,Z 369.111,A -85,B 0,C 180,E1 -8108.776,E2 -8108.776} C_VEL
LIN {X 0,Y 460.625,Z 369.107,A -85,B 0,C 180,E1 -8112.457,E2 -8112.457} C_VEL
LIN {X 0,Y 460.591,Z 369.108,A -85,B 0,C 180,E1 -8115.998,E2 -8115.998} C_VEL
LIN {X 0,Y 460.563,Z 369.116,A -85,B 0,C 180,E1 -8118.902,E2 -8118.902} C_VEL
LIN {X 0,Y 460.511,Z 369.117,A -85,B 0,C 180,E1 -8121.486,E2 -8121.486} C_VEL
LIN {X 0,Y 460.537,Z 369.118,A -85,B 0,C 180,E1 -8124.333,E2 -8124.333} C_VEL
LIN {X 0,Y 460.577,Z 369.11,A -85,B 0,C 180,E1 -8127.244,E2 -8127.244} C_VEL
LIN {X 0,Y 460.504,Z 369.122,A -85,B 0,C 180,E1 -8130.241,E2 -8130.241} C_VEL
LIN {X 0,Y 460.523,Z 369.116,A -85,B 0,C 180,E1 -8133.326,E2 -8133.326} C_VEL
LIN {X 0,Y 460.473,Z 369.129,A -85,B 0,C 180,E1 -8136.53,E2 -8136.53} C_VEL
LIN {X 0,Y 460.57,Z 369.112,A -85,B 0,C 180,E1 -8139.859,E2 -8139.859} C_VEL
LIN {X 0,Y 460.538,Z 369.115,A -85,B 0,C 180,E1 -8142.905,E2 -8142.905} C_VEL
LIN {X 0,Y 460.508,Z 369.12,A -85,B 0,C 180,E1 -8145.831,E2 -8145.831} C_VEL
LIN {X 0,Y 460.528,Z 369.116,A -85,B 0,C 180,E1 -8148.99,E2 -8148.99} C_VEL
LIN {X 0,Y 460.524,Z 369.115,A -85,B 0,C 180,E1 -8151.268,E2 -8151.268} C_VEL
LIN {X 0,Y 460.512,Z 369.12,A -85,B 0,C 180,E1 -8154.556,E2 -8154.556} C_VEL
LIN {X 0,Y 460.531,Z 369.117,A -85,B 0,C 180,E1 -8157.716,E2 -8157.716} C_VEL
LIN {X 0,Y 460.541,Z 369.114,A -85,B 0,C 180,E1 -8160.77,E2 -8160.77} C_VEL
LIN {X 0,Y 460.556,Z 369.115,A -85,B 0,C 180,E1 -8163.735,E2 -8163.735} C_VEL
LIN {X 0,Y 460.545,Z 369.119,A -85,B 0,C 180,E1 -8166.625,E2 -8166.625} C_VEL
LIN {X 0,Y 460.55,Z 369.139,A -85,B 0,C 180,E1 -8168.57,E2 -8168.57} C_VEL
LIN {X 0,Y 461.942,Z 377.001,A -85,B 0,C 180,E1 -8170.446,E2 -8170.446} C_VEL
LIN {X 0,Y 461.577,Z 387.525,A -85,B 0,C 180,E1 -8172.781,E2 -8172.781} C_VEL
LIN {X 0,Y 464.608,Z 403.313,A -85,B 0,C 180,E1 -8173.157,E2 -8173.157} C_VEL
LIN {X 0,Y 464.425,Z 433.815,A -85,B 0,C 180,E1 -8173.633,E2 -8173.633} C_VEL
LIN {X 0,Y 463.683,Z 439.661,A -85,B 0,C 180,E1 -8173.698,E2 -8173.698} C_VEL
LIN {X 0,Y 458.043,Z 458.668,A -85,B 0,C 180,E1 -8173.792,E2 -8173.792} C_VEL
LIN {X 0,Y 457.368,Z 464.511,A -85,B 0,C 180,E1 -8173.861,E2 -8173.861} C_VEL
LIN {X 0,Y 457.068,Z 494.891,A -85,B 0,C 180,E1 -8174.362,E2 -8174.362} C_VEL
LIN {X 0,Y 456.668,Z 508.748,A -85,B 0,C 180,E1 -8174.777,E2 -8174.777} C_VEL
LIN {X 0,Y 456.299,Z 521.142,A -85,B 0,C 180,E1 -8175.335,E2 -8175.335} C_VEL
LIN {X 0,Y 455.828,Z 532.99,A -85,B 0,C 180,E1 -8176.061,E2 -8176.061} C_VEL
LIN {X 0,Y 455.324,Z 544.337,A -85,B 0,C 180,E1 -8176.954,E2 -8176.954} C_VEL
LIN {X 0,Y 454.703,Z 554.569,A -85,B 0,C 180,E1 -8177.956,E2 -8177.956} C_VEL
LIN {X 0,Y 454.226,Z 563.742,A -85,B 0,C 180,E1 -8179.074,E2 -8179.074} C_VEL
LIN {X 0,Y 453.703,Z 572.647,A -85,B 0,C 180,E1 -8180.415,E2 -8180.415} C_VEL
LIN {X 0,Y 453.251,Z 579.816,A -85,B 0,C 180,E1 -8181.754,E2 -8181.754} C_VEL
LIN {X 0,Y 452.961,Z 585.996,A -85,B 0,C 180,E1 -8183.221,E2 -8183.221} C_VEL
LIN {X 0,Y 452.703,Z 590.66,A -85,B 0,C 180,E1 -8184.655,E2 -8184.655} C_VEL
LIN {X 0,Y 452.638,Z 592.941,A -85,B 0,C 180,E1 -8185.548,E2 -8185.548} C_VEL
LIN {X 0,Y 452.652,Z 594.796,A -85,B 0,C 180,E1 -8186.439,E2 -8186.439} C_VEL
LIN {X 0,Y 452.552,Z 596.199,A -85,B 0,C 180,E1 -8187.33,E2 -8187.33} C_VEL
LIN {X 0,Y 452.459,Z 597.809,A -85,B 0,C 180,E1 -8189.11,E2 -8189.11} C_VEL
LIN {X 0,Y 452.466,Z 598.043,A -85,B 0,C 180,E1 -8190,E2 -8190} C_VEL
LIN {X 0,Y 452.459,Z 597.857,A -85,B 0,C 180,E1 -8190.89,E2 -8190.89} C_VEL
LIN {X 0,Y 452.552,Z 596.31,A -85,B 0,C 180,E1 -8192.67,E2 -8192.67} C_VEL
LIN {X 0,Y 452.652,Z 594.956,A -85,B 0,C 180,E1 -8193.561,E2 -8193.561} C_VEL
LIN {X 0,Y 452.632,Z 592.103,A -85,B 0,C 180,E1 -8194.899,E2 -8194.899} C_VEL
LIN {X 0,Y 452.907,Z 588.223,A -85,B 0,C 180,E1 -8196.236,E2 -8196.236} C_VEL
LIN {X 0,Y 453.077,Z 583.224,A -85,B 0,C 180,E1 -8197.576,E2 -8197.576} C_VEL
LIN {X 0,Y 453.403,Z 576.928,A -85,B 0,C 180,E1 -8198.917,E2 -8198.917} C_VEL
LIN {X 0,Y 453.862,Z 569.042,A -85,B 0,C 180,E1 -8200.257,E2 -8200.257} C_VEL
LIN {X 0,Y 454.274,Z 561.003,A -85,B 0,C 180,E1 -8201.376,E2 -8201.376} C_VEL
LIN {X 0,Y 454.942,Z 551.184,A -85,B 0,C 180,E1 -8202.49,E2 -8202.49} C_VEL
LIN {X 0,Y 455.484,Z 540.009,A -85,B 0,C 180,E1 -8203.507,E2 -8203.507} C_VEL
LIN {X 0,Y 455.982,Z 529.322,A -85,B 0,C 180,E1 -8204.276,E2 -8204.276} C_VEL
LIN {X 0,Y 456.4,Z 517.367,A -85,B 0,C 180,E1 -8204.947,E2 -8204.947} C_VEL
LIN {X 0,Y 456.853,Z 504.247,A -85,B 0,C 180,E1 -8205.474,E2 -8205.474} C_VEL
LIN {X 0,Y 457.077,Z 491.053,A -85,B 0,C 180,E1 -8205.809,E2 -8205.809} C_VEL
LIN {X 0,Y 457.728,Z 403.164,A -85,B 0,C 180,E1 -8207.204,E2 -8207.204} C_VEL
LIN {X 0,Y 454.64,Z 387.814,A -85,B 0,C 180,E1 -8207.579,E2 -8207.579} C_VEL
LIN {X 0,Y 454.964,Z 377.637,A -85,B 0,C 180,E1 -8209.867,E2 -8209.867} C_VEL
LIN {X 0,Y 453.463,Z 370.006,A -85,B 0,C 180,E1 -8211.726,E2 -8211.726} C_VEL
LIN {X 0,Y 453.515,Z 369.995,A -85,B 0,C 180,E1 -8214.734,E2 -8214.734} C_VEL
LIN {X 0,Y 453.532,Z 369.994,A -85,B 0,C 180,E1 -8217.959,E2 -8217.959} C_VEL
LIN {X 0,Y 453.466,Z 369.998,A -85,B 0,C 180,E1 -8221.524,E2 -8221.524} C_VEL
LIN {X 0,Y 453.488,Z 369.992,A -85,B 0,C 180,E1 -8224.777,E2 -8224.777} C_VEL
LIN {X 0,Y 453.471,Z 369.996,A -85,B 0,C 180,E1 -8228.31,E2 -8228.31} C_VEL
LIN {X 0,Y 453.491,Z 369.992,A -85,B 0,C 180,E1 -8230.608,E2 -8230.608} C_VEL
LIN {X 0,Y 453.452,Z 369.998,A -85,B 0,C 180,E1 -8233.243,E2 -8233.243} C_VEL
LIN {X 0,Y 453.473,Z 370.001,A -85,B 0,C 180,E1 -8235.78,E2 -8235.78} C_VEL
LIN {X 0,Y 453.492,Z 369.993,A -85,B 0,C 180,E1 -8238.21,E2 -8238.21} C_VEL
LIN {X 0,Y 453.521,Z 369.988,A -85,B 0,C 180,E1 -8240.788,E2 -8240.788} C_VEL
LIN {X 0,Y 453.452,Z 370.001,A -85,B 0,C 180,E1 -8243.917,E2 -8243.917} C_VEL
LIN {X 0,Y 453.481,Z 369.996,A -85,B 0,C 180,E1 -8247.151,E2 -8247.151} C_VEL
LIN {X 0,Y 453.468,Z 369.995,A -85,B 0,C 180,E1 -8250.268,E2 -8250.268} C_VEL
LIN {X 0,Y 453.507,Z 369.995,A -85,B 0,C 180,E1 -8253.294,E2 -8253.294} C_VEL
LIN {X 0,Y 453.497,Z 369.991,A -85,B 0,C 180,E1 -8256.238,E2 -8256.238} C_VEL
LIN {X 0,Y 453.486,Z 369.997,A -85,B 0,C 180,E1 -8259.118,E2 -8259.118} C_VEL
LIN {X 0,Y 453.504,Z 369.991,A -85,B 0,C 180,E1 -8261.944,E2 -8261.944} C_VEL
LIN {X 0,Y 453.533,Z 369.988,A -85,B 0,C 180,E1 -8264.726,E2 -8264.726} C_VEL
LIN {X 0,Y 453.593,Z 369.984,A -85,B 0,C 180,E1 -8267.472,E2 -8267.472} C_VEL
LIN {X 0,Y 453.585,Z 369.986,A -85,B 0,C 180,E1 -8271.086,E2 -8271.086} C_VEL
LIN {X 0,Y 453.669,Z 369.971,A -85,B 0,C 180,E1 -8273.775,E2 -8273.775} C_VEL
LIN {X 0,Y 453.758,Z 369.964,A -85,B 0,C 180,E1 -8277.337,E2 -8277.337} C_VEL
LIN {X 0,Y 453.815,Z 369.951,A -85,B 0,C 180,E1 -8280,E2 -8280} C_VEL
LIN {X 0,Y 453.759,Z 369.961,A -85,B 0,C 180,E1 -8282.663,E2 -8282.663} C_VEL
LIN {X 0,Y 453.671,Z 369.969,A -85,B 0,C 180,E1 -8286.225,E2 -8286.225} C_VEL
LIN {X 0,Y 453.585,Z 369.987,A -85,B 0,C 180,E1 -8288.913,E2 -8288.913} C_VEL
LIN {X 0,Y 453.593,Z 369.982,A -85,B 0,C 180,E1 -8292.551,E2 -8292.551} C_VEL
LIN {X 0,Y 453.536,Z 369.987,A -85,B 0,C 180,E1 -8296.196,E2 -8296.196} C_VEL
LIN {X 0,Y 453.512,Z 369.994,A -85,B 0,C 180,E1 -8299.041,E2 -8299.041} C_VEL
LIN {X 0,Y 453.471,Z 369.994,A -85,B 0,C 180,E1 -8301.836,E2 -8301.836} C_VEL
LIN {X 0,Y 453.508,Z 369.998,A -85,B 0,C 180,E1 -8304.735,E2 -8304.735} C_VEL
LIN {X 0,Y 453.53,Z 369.987,A -85,B 0,C 180,E1 -8307.962,E2 -8307.962} C_VEL
LIN {X 0,Y 453.46,Z 369.996,A -85,B 0,C 180,E1 -8311.526,E2 -8311.526} C_VEL
LIN {X 0,Y 453.483,Z 369.998,A -85,B 0,C 180,E1 -8314.778,E2 -8314.778} C_VEL
LIN {X 0,Y 453.478,Z 369.998,A -85,B 0,C 180,E1 -8318.31,E2 -8318.31} C_VEL
LIN {X 0,Y 453.511,Z 369.996,A -85,B 0,C 180,E1 -8320.607,E2 -8320.607} C_VEL
LIN {X 0,Y 453.477,Z 369.994,A -85,B 0,C 180,E1 -8323.248,E2 -8323.248} C_VEL
LIN {X 0,Y 453.469,Z 369.995,A -85,B 0,C 180,E1 -8325.781,E2 -8325.781} C_VEL
LIN {X 0,Y 453.478,Z 369.998,A -85,B 0,C 180,E1 -8328.21,E2 -8328.21} C_VEL
LIN {X 0,Y 453.513,Z 369.992,A -85,B 0,C 180,E1 -8330.791,E2 -8330.791} C_VEL
LIN {X 0,Y 453.455,Z 369.999,A -85,B 0,C 180,E1 -8333.918,E2 -8333.918} C_VEL
LIN {X 0,Y 453.482,Z 369.993,A -85,B 0,C 180,E1 -8337.152,E2 -8337.152} C_VEL
LIN {X 0,Y 453.475,Z 370.002,A -85,B 0,C 180,E1 -8340.269,E2 -8340.269} C_VEL
LIN {X 0,Y 453.59,Z 370.102,A -85,B 0,C 180,E1 -8343.346,E2 -8343.346} C_VEL
LIN {X 0,Y 456.071,Z 383.053,A -85,B 0,C 180,E1 -8345.91,E2 -8345.91} C_VEL
LIN {X 0,Y 455.704,Z 392.977,A -85,B 0,C 180,E1 -8347.72,E2 -8347.72} C_VEL
LIN {X 0,Y 454.703,Z 412.879,A -85,B 0,C 180,E1 -8351.294,E2 -8351.294} C_VEL
LIN {X 0,Y 454.407,Z 419.395,A -85,B 0,C 180,E1 -8352.444,E2 -8352.444} C_VEL
LIN {X 0,Y 457.611,Z 441.489,A -85,B 0,C 180,E1 -8352.924,E2 -8352.924} C_VEL
LIN {X 0,Y 456.858,Z 527.614,A -85,B 0,C 180,E1 -8354.297,E2 -8354.297} C_VEL
LIN {X 0,Y 456.476,Z 540.882,A -85,B 0,C 180,E1 -8354.684,E2 -8354.684} C_VEL
LIN {X 0,Y 455.953,Z 553.046,A -85,B 0,C 180,E1 -8355.209,E2 -8355.209} C_VEL
LIN {X 0,Y 455.393,Z 565.325,A -85,B 0,C 180,E1 -8355.933,E2 -8355.933} C_VEL
LIN {X 0,Y 454.712,Z 577.099,A -85,B 0,C 180,E1 -8356.837,E2 -8356.837} C_VEL
LIN {X 0,Y 454.286,Z 587.391,A -85,B 0,C 180,E1 -8357.832,E2 -8357.832} C_VEL
LIN {X 0,Y 453.806,Z 595.942,A -85,B 0,C 180,E1 -8358.838,E2 -8358.838} C_VEL
LIN {X 0,Y 453.355,Z 603.833,A -85,B 0,C 180,E1 -8359.957,E2 -8359.957} C_VEL
LIN {X 0,Y 453.001,Z 611.544,A -85,B 0,C 180,E1 -8361.3,E2 -8361.3} C_VEL
LIN {X 0,Y 452.719,Z 618.656,A -85,B 0,C 180,E1 -8362.866,E2 -8362.866} C_VEL
LIN {X 0,Y 452.558,Z 623.388,A -85,B 0,C 180,E1 -8364.207,E2 -8364.207} C_VEL
LIN {X 0,Y 452.487,Z 627.005,A -85,B 0,C 180,E1 -8365.546,E2 -8365.546} C_VEL
LIN {X 0,Y 452.483,Z 628.872,A -85,B 0,C 180,E1 -8366.438,E2 -8366.438} C_VEL
LIN {X 0,Y 452.508,Z 630.273,A -85,B 0,C 180,E1 -8367.329,E2 -8367.329} C_VEL
LIN {X 0,Y 452.457,Z 631.88,A -85,B 0,C 180,E1 -8369.11,E2 -8369.11} C_VEL
LIN {X 0,Y 452.464,Z 632.097,A -85,B 0,C 180,E1 -8370,E2 -8370} C_VEL
LIN {X 0,Y 452.457,Z 631.88,A -85,B 0,C 180,E1 -8370.89,E2 -8370.89} C_VEL
LIN {X 0,Y 452.508,Z 630.275,A -85,B 0,C 180,E1 -8372.671,E2 -8372.671} C_VEL
LIN {X 0,Y 452.483,Z 628.874,A -85,B 0,C 180,E1 -8373.562,E2 -8373.562} C_VEL
LIN {X 0,Y 452.546,Z 625.931,A -85,B 0,C 180,E1 -8374.9,E2 -8374.9} C_VEL
LIN {X 0,Y 452.61,Z 621.408,A -85,B 0,C 180,E1 -8376.396,E2 -8376.396} C_VEL
LIN {X 0,Y 452.804,Z 615.823,A -85,B 0,C 180,E1 -8377.805,E2 -8377.805} C_VEL
LIN {X 0,Y 453.089,Z 609.132,A -85,B 0,C 180,E1 -8379.148,E2 -8379.148} C_VEL
LIN {X 0,Y 453.482,Z 600.834,A -85,B 0,C 180,E1 -8380.492,E2 -8380.492} C_VEL
LIN {X 0,Y 454.008,Z 592.335,A -85,B 0,C 180,E1 -8381.609,E2 -8381.609} C_VEL
LIN {X 0,Y 454.518,Z 582.704,A -85,B 0,C 180,E1 -8382.645,E2 -8382.645} C_VEL
LIN {X 0,Y 455.093,Z 571.445,A -85,B 0,C 180,E1 -8383.621,E2 -8383.621} C_VEL
LIN {X 0,Y 455.631,Z 560.06,A -85,B 0,C 180,E1 -8384.402,E2 -8384.402} C_VEL
LIN {X 0,Y 456.169,Z 548.385,A -85,B 0,C 180,E1 -8385.012,E2 -8385.012} C_VEL
LIN {X 0,Y 456.631,Z 535.85,A -85,B 0,C 180,E1 -8385.482,E2 -8385.482} C_VEL
LIN {X 0,Y 456.951,Z 523.159,A -85,B 0,C 180,E1 -8385.785,E2 -8385.785} C_VEL
LIN {X 0,Y 457.535,Z 439.649,A -85,B 0,C 180,E1 -8387.106,E2 -8387.106} C_VEL
LIN {X 0,Y 454.413,Z 419.273,A -85,B 0,C 180,E1 -8387.557,E2 -8387.557} C_VEL
LIN {X 0,Y 455.247,Z 401.188,A -85,B 0,C 180,E1 -8390.797,E2 -8390.797} C_VEL
LIN {X 0,Y 456.091,Z 385.579,A -85,B 0,C 180,E1 -8393.618,E2 -8393.618} C_VEL
LIN {X 0,Y 455.734,Z 380.838,A -85,B 0,C 180,E1 -8394.514,E2 -8394.514} C_VEL
LIN {X 0,Y 453.576,Z 369.985,A -85,B 0,C 180,E1 -8396.701,E2 -8396.701} C_VEL
LIN {X 0,Y 453.472,Z 370.002,A -85,B 0,C 180,E1 -8399.784,E2 -8399.784} C_VEL
LIN {X 0,Y 453.49,Z 369.994,A -85,B 0,C 180,E1 -8403.189,E2 -8403.189} C_VEL
LIN {X 0,Y 453.454,Z 369.997,A -85,B 0,C 180,E1 -8406.299,E2 -8406.299} C_VEL
LIN {X 0,Y 453.514,Z 369.994,A -85,B 0,C 180,E1 -8409.446,E2 -8409.446} C_VEL
LIN {X 0,Y 453.464,Z 369.996,A -85,B 0,C 180,E1 -8412.994,E2 -8412.994} C_VEL
LIN {X 0,Y 453.473,Z 369.999,A -85,B 0,C 180,E1 -8415.78,E2 -8415.78} C_VEL
LIN {X 0,Y 453.492,Z 369.992,A -85,B 0,C 180,E1 -8418.211,E2 -8418.211} C_VEL
LIN {X 0,Y 453.525,Z 369.988,A -85,B 0,C 180,E1 -8420.787,E2 -8420.787} C_VEL
LIN {X 0,Y 453.451,Z 369.999,A -85,B 0,C 180,E1 -8423.917,E2 -8423.917} C_VEL
LIN {X 0,Y 453.477,Z 369.998,A -85,B 0,C 180,E1 -8427.151,E2 -8427.151} C_VEL
LIN {X 0,Y 453.507,Z 369.99,A -85,B 0,C 180,E1 -8430.271,E2 -8430.271} C_VEL
LIN {X 0,Y 453.522,Z 369.996,A -85,B 0,C 180,E1 -8433.295,E2 -8433.295} C_VEL
LIN {X 0,Y 453.497,Z 369.991,A -85,B 0,C 180,E1 -8436.238,E2 -8436.238} C_VEL
LIN {X 0,Y 453.486,Z 369.999,A -85,B 0,C 180,E1 -8439.118,E2 -8439.118} C_VEL
LIN {X 0,Y 453.503,Z 369.991,A -85,B 0,C 180,E1 -8441.944,E2 -8441.944} C_VEL
LIN {X 0,Y 453.532,Z 369.989,A -85,B 0,C 180,E1 -8444.726,E2 -8444.726} C_VEL
LIN {X 0,Y 453.593,Z 369.982,A -85,B 0,C 180,E1 -8447.472,E2 -8447.472} C_VEL
LIN {X 0,Y 453.585,Z 369.988,A -85,B 0,C 180,E1 -8451.086,E2 -8451.086} C_VEL
LIN {X 0,Y 453.669,Z 369.97,A -85,B 0,C 180,E1 -8453.775,E2 -8453.775} C_VEL
LIN {X 0,Y 453.758,Z 369.962,A -85,B 0,C 180,E1 -8457.337,E2 -8457.337} C_VEL
LIN {X 0,Y 453.815,Z 369.951,A -85,B 0,C 180,E1 -8460,E2 -8460} C_VEL
LIN {X 0,Y 453.758,Z 369.963,A -85,B 0,C 180,E1 -8462.663,E2 -8462.663} C_VEL
LIN {X 0,Y 453.671,Z 369.97,A -85,B 0,C 180,E1 -8466.225,E2 -8466.225} C_VEL
LIN {X 0,Y 453.585,Z 369.987,A -85,B 0,C 180,E1 -8468.914,E2 -8468.914} C_VEL
LIN {X 0,Y 453.593,Z 369.984,A -85,B 0,C 180,E1 -8472.551,E2 -8472.551} C_VEL
LIN {X 0,Y 453.536,Z 369.988,A -85,B 0,C 180,E1 -8476.196,E2 -8476.196} C_VEL
LIN {X 0,Y 453.512,Z 369.992,A -85,B 0,C 180,E1 -8479.041,E2 -8479.041} C_VEL
LIN {X 0,Y 453.471,Z 369.994,A -85,B 0,C 180,E1 -8481.837,E2 -8481.837} C_VEL
LIN {X 0,Y 453.508,Z 369.996,A -85,B 0,C 180,E1 -8484.735,E2 -8484.735} C_VEL
LIN {X 0,Y 453.531,Z 369.988,A -85,B 0,C 180,E1 -8487.962,E2 -8487.962} C_VEL
LIN {X 0,Y 453.46,Z 369.995,A -85,B 0,C 180,E1 -8491.526,E2 -8491.526} C_VEL
LIN {X 0,Y 453.483,Z 369.997,A -85,B 0,C 180,E1 -8494.778,E2 -8494.778} C_VEL
LIN {X 0,Y 453.476,Z 370,A -85,B 0,C 180,E1 -8498.311,E2 -8498.311} C_VEL
LIN {X 0,Y 453.512,Z 369.994,A -85,B 0,C 180,E1 -8500.607,E2 -8500.607} C_VEL
LIN {X 0,Y 453.478,Z 369.993,A -85,B 0,C 180,E1 -8503.248,E2 -8503.248} C_VEL
LIN {X 0,Y 453.463,Z 369.997,A -85,B 0,C 180,E1 -8505.78,E2 -8505.78} C_VEL
LIN {X 0,Y 453.476,Z 370.001,A -85,B 0,C 180,E1 -8508.21,E2 -8508.21} C_VEL
LIN {X 0,Y 453.513,Z 369.991,A -85,B 0,C 180,E1 -8510.791,E2 -8510.791} C_VEL
LIN {X 0,Y 453.456,Z 370,A -85,B 0,C 180,E1 -8513.918,E2 -8513.918} C_VEL
LIN {X 0,Y 453.482,Z 369.993,A -85,B 0,C 180,E1 -8517.152,E2 -8517.152} C_VEL
LIN {X 0,Y 453.476,Z 370,A -85,B 0,C 180,E1 -8520.269,E2 -8520.269} C_VEL
LIN {X 0,Y 453.505,Z 369.99,A -85,B 0,C 180,E1 -8523.295,E2 -8523.295} C_VEL
LIN {X 0,Y 453.499,Z 369.999,A -85,B 0,C 180,E1 -8526.239,E2 -8526.239} C_VEL
LIN {X 0,Y 453.52,Z 370.141,A -85,B 0,C 180,E1 -8528.403,E2 -8528.403} C_VEL
LIN {X 0,Y 455,Z 378.514,A -85,B 0,C 180,E1 -8530.428,E2 -8530.428} C_VEL
LIN {X 0,Y 454.644,Z 387.794,A -85,B 0,C 180,E1 -8532.513,E2 -8532.513} C_VEL
LIN {X 0,Y 457.82,Z 403.633,A -85,B 0,C 180,E1 -8532.9,E2 -8532.9} C_VEL
LIN {X 0,Y 457.368,Z 464.511,A -85,B 0,C 180,E1 -8533.861,E2 -8533.861} C_VEL
LIN {X 0,Y 456.695,Z 470.359,A -85,B 0,C 180,E1 -8533.926,E2 -8533.926} C_VEL
LIN {X 0,Y 451.023,Z 489.355,A -85,B 0,C 180,E1 -8534.02,E2 -8534.02} C_VEL
LIN {X 0,Y 450.25,Z 495.162,A -85,B 0,C 180,E1 -8534.119,E2 -8534.119} C_VEL
LIN {X 0,Y 449.833,Z 509.026,A -85,B 0,C 180,E1 -8534.54,E2 -8534.54} C_VEL
LIN {X 0,Y 449.428,Z 521.418,A -85,B 0,C 180,E1 -8535.106,E2 -8535.106} C_VEL
LIN {X 0,Y 448.953,Z 533.262,A -85,B 0,C 180,E1 -8535.843,E2 -8535.843} C_VEL
LIN {X 0,Y 448.402,Z 544.711,A -85,B 0,C 180,E1 -8536.758,E2 -8536.758} C_VEL
LIN {X 0,Y 447.757,Z 554.84,A -85,B 0,C 180,E1 -8537.767,E2 -8537.767} C_VEL
LIN {X 0,Y 447.25,Z 564.013,A -85,B 0,C 180,E1 -8538.902,E2 -8538.902} C_VEL
LIN {X 0,Y 446.687,Z 572.918,A -85,B 0,C 180,E1 -8540.263,E2 -8540.263} C_VEL
LIN {X 0,Y 446.218,Z 580.086,A -85,B 0,C 180,E1 -8541.623,E2 -8541.623} C_VEL
LIN {X 0,Y 445.971,Z 584.919,A -85,B 0,C 180,E1 -8542.758,E2 -8542.758} C_VEL
LIN {X 0,Y 445.8,Z 589.612,A -85,B 0,C 180,E1 -8544.119,E2 -8544.119} C_VEL
LIN {X 0,Y 445.549,Z 593.21,A -85,B 0,C 180,E1 -8545.477,E2 -8545.477} C_VEL
LIN {X 0,Y 445.57,Z 595.064,A -85,B 0,C 180,E1 -8546.383,E2 -8546.383} C_VEL
LIN {X 0,Y 445.481,Z 596.466,A -85,B 0,C 180,E1 -8547.287,E2 -8547.287} C_VEL
LIN {X 0,Y 445.368,Z 598.076,A -85,B 0,C 180,E1 -8549.096,E2 -8549.096} C_VEL
LIN {X 0,Y 445.372,Z 598.31,A -85,B 0,C 180,E1 -8550,E2 -8550} C_VEL
LIN {X 0,Y 445.368,Z 598.124,A -85,B 0,C 180,E1 -8550.904,E2 -8550.904} C_VEL
LIN {X 0,Y 445.481,Z 596.576,A -85,B 0,C 180,E1 -8552.713,E2 -8552.713} C_VEL
LIN {X 0,Y 445.57,Z 595.223,A -85,B 0,C 180,E1 -8553.617,E2 -8553.617} C_VEL
LIN {X 0,Y 445.565,Z 592.369,A -85,B 0,C 180,E1 -8554.977,E2 -8554.977} C_VEL
LIN {X 0,Y 445.845,Z 588.489,A -85,B 0,C 180,E1 -8556.335,E2 -8556.335} C_VEL
LIN {X 0,Y 446.026,Z 583.49,A -85,B 0,C 180,E1 -8557.697,E2 -8557.697} C_VEL
LIN {X 0,Y 446.406,Z 577.192,A -85,B 0,C 180,E1 -8559.058,E2 -8559.058} C_VEL
LIN {X 0,Y 446.877,Z 569.306,A -85,B 0,C 180,E1 -8560.42,E2 -8560.42} C_VEL
LIN {X 0,Y 447.333,Z 561.266,A -85,B 0,C 180,E1 -8561.555,E2 -8561.555} C_VEL
LIN {X 0,Y 448.027,Z 551.446,A -85,B 0,C 180,E1 -8562.686,E2 -8562.686} C_VEL
LIN {X 0,Y 448.509,Z 541.789,A -85,B 0,C 180,E1 -8563.594,E2 -8563.594} C_VEL
LIN {X 0,Y 449.014,Z 531.341,A -85,B 0,C 180,E1 -8564.387,E2 -8564.387} C_VEL
LIN {X 0,Y 449.533,Z 518.75,A -85,B 0,C 180,E1 -8565.123,E2 -8565.123} C_VEL
LIN {X 0,Y 449.977,Z 506.152,A -85,B 0,C 180,E1 -8565.658,E2 -8565.658} C_VEL
LIN {X 0,Y 450.259,Z 492.799,A -85,B 0,C 180,E1 -8566.026,E2 -8566.026} C_VEL
LIN {X 0,Y 451.022,Z 404.435,A -85,B 0,C 180,E1 -8567.451,E2 -8567.451} C_VEL
LIN {X 0,Y 447.711,Z 388.05,A -85,B 0,C 180,E1 -8567.865,E2 -8567.865} C_VEL
LIN {X 0,Y 448.077,Z 379.683,A -85,B 0,C 180,E1 -8569.764,E2 -8569.764} C_VEL
LIN {X 0,Y 446.427,Z 370.884,A -85,B 0,C 180,E1 -8571.956,E2 -8571.956} C_VEL
LIN {X 0,Y 446.459,Z 370.874,A -85,B 0,C 180,E1 -8575.152,E2 -8575.152} C_VEL
LIN {X 0,Y 446.485,Z 370.87,A -85,B 0,C 180,E1 -8578.178,E2 -8578.178} C_VEL
LIN {X 0,Y 446.419,Z 370.878,A -85,B 0,C 180,E1 -8581.774,E2 -8581.774} C_VEL
LIN {X 0,Y 446.429,Z 370.872,A -85,B 0,C 180,E1 -8584.522,E2 -8584.522} C_VEL
LIN {X 0,Y 446.429,Z 370.876,A -85,B 0,C 180,E1 -8588.081,E2 -8588.081} C_VEL
LIN {X 0,Y 446.424,Z 370.872,A -85,B 0,C 180,E1 -8590.917,E2 -8590.917} C_VEL
LIN {X 0,Y 446.414,Z 370.88,A -85,B 0,C 180,E1 -8593.843,E2 -8593.843} C_VEL
LIN {X 0,Y 446.443,Z 370.871,A -85,B 0,C 180,E1 -8596.396,E2 -8596.396} C_VEL
LIN {X 0,Y 446.463,Z 370.873,A -85,B 0,C 180,E1 -8599.804,E2 -8599.804} C_VEL
LIN {X 0,Y 446.427,Z 370.874,A -85,B 0,C 180,E1 -8602.123,E2 -8602.123} C_VEL
LIN {X 0,Y 446.426,Z 370.878,A -85,B 0,C 180,E1 -8605.476,E2 -8605.476} C_VEL
LIN {X 0,Y 446.41,Z 370.874,A -85,B 0,C 180,E1 -8608.699,E2 -8608.699} C_VEL
LIN {X 0,Y 446.478,Z 370.869,A -85,B 0,C 180,E1 -8611.821,E2 -8611.821} C_VEL
LIN {X 0,Y 446.452,Z 370.87,A -85,B 0,C 180,E1 -8614.847,E2 -8614.847} C_VEL
LIN {X 0,Y 446.442,Z 370.87,A -85,B 0,C 180,E1 -8618.244,E2 -8618.244} C_VEL
LIN {X 0,Y 446.45,Z 370.873,A -85,B 0,C 180,E1 -8621.649,E2 -8621.649} C_VEL
LIN {X 0,Y 446.5,Z 370.863,A -85,B 0,C 180,E1 -8624.479,E2 -8624.479} C_VEL
LIN {X 0,Y 446.532,Z 370.859,A -85,B 0,C 180,E1 -8628.193,E2 -8628.193} C_VEL
LIN {X 0,Y 446.592,Z 370.852,A -85,B 0,C 180,E1 -8631.858,E2 -8631.858} C_VEL
LIN {X 0,Y 446.638,Z 370.847,A -85,B 0,C 180,E1 -8634.582,E2 -8634.582} C_VEL
LIN {X 0,Y 446.702,Z 370.843,A -85,B 0,C 180,E1 -8637.295,E2 -8637.295} C_VEL
LIN {X 0,Y 446.785,Z 370.827,A -85,B 0,C 180,E1 -8640,E2 -8640} C_VEL
LIN {X 0,Y 446.703,Z 370.841,A -85,B 0,C 180,E1 -8642.705,E2 -8642.705} C_VEL
LIN {X 0,Y 446.64,Z 370.846,A -85,B 0,C 180,E1 -8646.324,E2 -8646.324} C_VEL
LIN {X 0,Y 446.531,Z 370.866,A -85,B 0,C 180,E1 -8649.055,E2 -8649.055} C_VEL
LIN {X 0,Y 446.526,Z 370.865,A -85,B 0,C 180,E1 -8652.73,E2 -8652.73} C_VEL
LIN {X 0,Y 446.482,Z 370.868,A -85,B 0,C 180,E1 -8656.459,E2 -8656.459} C_VEL
LIN {X 0,Y 446.461,Z 370.87,A -85,B 0,C 180,E1 -8659.304,E2 -8659.304} C_VEL
LIN {X 0,Y 446.413,Z 370.875,A -85,B 0,C 180,E1 -8662.2,E2 -8662.2} C_VEL
LIN {X 0,Y 446.451,Z 370.871,A -85,B 0,C 180,E1 -8665.153,E2 -8665.153} C_VEL
LIN {X 0,Y 446.477,Z 370.867,A -85,B 0,C 180,E1 -8668.179,E2 -8668.179} C_VEL
LIN {X 0,Y 446.413,Z 370.873,A -85,B 0,C 180,E1 -8671.776,E2 -8671.776} C_VEL
LIN {X 0,Y 446.425,Z 370.879,A -85,B 0,C 180,E1 -8674.523,E2 -8674.523} C_VEL
LIN {X 0,Y 446.432,Z 370.873,A -85,B 0,C 180,E1 -8678.084,E2 -8678.084} C_VEL
LIN {X 0,Y 446.442,Z 370.873,A -85,B 0,C 180,E1 -8680.921,E2 -8680.921} C_VEL
LIN {X 0,Y 446.441,Z 370.871,A -85,B 0,C 180,E1 -8683.841,E2 -8683.841} C_VEL
LIN {X 0,Y 446.417,Z 370.88,A -85,B 0,C 180,E1 -8686.401,E2 -8686.401} C_VEL
LIN {X 0,Y 446.448,Z 370.87,A -85,B 0,C 180,E1 -8689.804,E2 -8689.804} C_VEL
LIN {X 0,Y 446.425,Z 370.877,A -85,B 0,C 180,E1 -8692.124,E2 -8692.124} C_VEL
LIN {X 0,Y 446.429,Z 370.872,A -85,B 0,C 180,E1 -8695.478,E2 -8695.478} C_VEL
LIN {X 0,Y 446.416,Z 370.879,A -85,B 0,C 180,E1 -8698.7,E2 -8698.7} C_VEL
LIN {X 0,Y 446.484,Z 370.872,A -85,B 0,C 180,E1 -8701.822,E2 -8701.822} C_VEL
LIN {X 0,Y 446.532,Z 370.96,A -85,B 0,C 180,E1 -8703.101,E2 -8703.101} C_VEL
LIN {X 0,Y 449.02,Z 383.564,A -85,B 0,C 180,E1 -8705.648,E2 -8705.648} C_VEL
LIN {X 0,Y 449.064,Z 389.276,A -85,B 0,C 180,E1 -8706.724,E2 -8706.724} C_VEL
LIN {X 0,Y 447.896,Z 409.522,A -85,B 0,C 180,E1 -8710.429,E2 -8710.429} C_VEL
LIN {X 0,Y 447.446,Z 418.964,A -85,B 0,C 180,E1 -8712.152,E2 -8712.152} C_VEL
LIN {X 0,Y 450.827,Z 442.225,A -85,B 0,C 180,E1 -8712.675,E2 -8712.675} C_VEL
LIN {X 0,Y 450.035,Z 527.358,A -85,B 0,C 180,E1 -8714.053,E2 -8714.053} C_VEL
LIN {X 0,Y 449.647,Z 540.623,A -85,B 0,C 180,E1 -8714.446,E2 -8714.446} C_VEL
LIN {X 0,Y 449.095,Z 552.784,A -85,B 0,C 180,E1 -8714.978,E2 -8714.978} C_VEL
LIN {X 0,Y 448.5,Z 565.061,A -85,B 0,C 180,E1 -8715.712,E2 -8715.712} C_VEL
LIN {X 0,Y 447.855,Z 575.875,A -85,B 0,C 180,E1 -8716.546,E2 -8716.546} C_VEL
LIN {X 0,Y 447.338,Z 586.05,A -85,B 0,C 180,E1 -8717.525,E2 -8717.525} C_VEL
LIN {X 0,Y 446.826,Z 595.676,A -85,B 0,C 180,E1 -8718.662,E2 -8718.662} C_VEL
LIN {X 0,Y 446.329,Z 603.566,A -85,B 0,C 180,E1 -8719.797,E2 -8719.797} C_VEL
LIN {X 0,Y 445.952,Z 611.277,A -85,B 0,C 180,E1 -8721.161,E2 -8721.161} C_VEL
LIN {X 0,Y 445.635,Z 618.388,A -85,B 0,C 180,E1 -8722.752,E2 -8722.752} C_VEL
LIN {X 0,Y 445.47,Z 622.616,A -85,B 0,C 180,E1 -8723.955,E2 -8723.955} C_VEL
LIN {X 0,Y 445.413,Z 626.739,A -85,B 0,C 180,E1 -8725.475,E2 -8725.475} C_VEL
LIN {X 0,Y 445.382,Z 628.605,A -85,B 0,C 180,E1 -8726.381,E2 -8726.381} C_VEL
LIN {X 0,Y 445.433,Z 630.007,A -85,B 0,C 180,E1 -8727.287,E2 -8727.287} C_VEL
LIN {X 0,Y 445.365,Z 631.614,A -85,B 0,C 180,E1 -8729.096,E2 -8729.096} C_VEL
LIN {X 0,Y 445.37,Z 631.831,A -85,B 0,C 180,E1 -8730,E2 -8730} C_VEL
LIN {X 0,Y 445.365,Z 631.613,A -85,B 0,C 180,E1 -8730.904,E2 -8730.904} C_VEL
LIN {X 0,Y 445.433,Z 630.008,A -85,B 0,C 180,E1 -8732.713,E2 -8732.713} C_VEL
LIN {X 0,Y 445.382,Z 628.606,A -85,B 0,C 180,E1 -8733.619,E2 -8733.619} C_VEL
LIN {X 0,Y 445.475,Z 625.664,A -85,B 0,C 180,E1 -8734.978,E2 -8734.978} C_VEL
LIN {X 0,Y 445.555,Z 620.242,A -85,B 0,C 180,E1 -8736.748,E2 -8736.748} C_VEL
LIN {X 0,Y 445.787,Z 614.539,A -85,B 0,C 180,E1 -8738.157,E2 -8738.157} C_VEL
LIN {X 0,Y 446.123,Z 607.623,A -85,B 0,C 180,E1 -8739.521,E2 -8739.521} C_VEL
LIN {X 0,Y 446.558,Z 598.974,A -85,B 0,C 180,E1 -8740.886,E2 -8740.886} C_VEL
LIN {X 0,Y 447.146,Z 590.111,A -85,B 0,C 180,E1 -8742.02,E2 -8742.02} C_VEL
LIN {X 0,Y 447.702,Z 579.616,A -85,B 0,C 180,E1 -8743.116,E2 -8743.116} C_VEL
LIN {X 0,Y 448.256,Z 569.743,A -85,B 0,C 180,E1 -8743.949,E2 -8743.949} C_VEL
LIN {X 0,Y 448.849,Z 557.862,A -85,B 0,C 180,E1 -8744.74,E2 -8744.74} C_VEL
LIN {X 0,Y 449.407,Z 545.506,A -85,B 0,C 180,E1 -8745.359,E2 -8745.359} C_VEL
LIN {X 0,Y 449.902,Z 532.827,A -85,B 0,C 180,E1 -8745.806,E2 -8745.806} C_VEL
LIN {X 0,Y 450.155,Z 519.573,A -85,B 0,C 180,E1 -8746.088,E2 -8746.088} C_VEL
LIN {X 0,Y 450.704,Z 440.054,A -85,B 0,C 180,E1 -8747.362,E2 -8747.362} C_VEL
LIN {X 0,Y 447.44,Z 418.992,A -85,B 0,C 180,E1 -8747.842,E2 -8747.842} C_VEL
LIN {X 0,Y 448.42,Z 399.64,A -85,B 0,C 180,E1 -8751.37,E2 -8751.37} C_VEL
LIN {X 0,Y 449.212,Z 385.34,A -85,B 0,C 180,E1 -8754.002,E2 -8754.002} C_VEL
LIN {X 0,Y 447.352,Z 374.843,A -85,B 0,C 180,E1 -8756.096,E2 -8756.096} C_VEL
LIN {X 0,Y 446.523,Z 370.865,A -85,B 0,C 180,E1 -8756.927,E2 -8756.927} C_VEL
LIN {X 0,Y 446.427,Z 370.878,A -85,B 0,C 180,E1 -8760.249,E2 -8760.249} C_VEL
LIN {X 0,Y 446.443,Z 370.874,A -85,B 0,C 180,E1 -8763.453,E2 -8763.453} C_VEL
LIN {X 0,Y 446.407,Z 370.874,A -85,B 0,C 180,E1 -8766.744,E2 -8766.744} C_VEL
LIN {X 0,Y 446.476,Z 370.872,A -85,B 0,C 180,E1 -8769.528,E2 -8769.528} C_VEL
LIN {X 0,Y 446.429,Z 370.871,A -85,B 0,C 180,E1 -8772.603,E2 -8772.603} C_VEL
LIN {X 0,Y 446.453,Z 370.871,A -85,B 0,C 180,E1 -8775.102,E2 -8775.102} C_VEL
LIN {X 0,Y 446.44,Z 370.87,A -85,B 0,C 180,E1 -8778.61,E2 -8778.61} C_VEL
LIN {X 0,Y 446.468,Z 370.869,A -85,B 0,C 180,E1 -8780.975,E2 -8780.975} C_VEL
LIN {X 0,Y 446.416,Z 370.873,A -85,B 0,C 180,E1 -8784.373,E2 -8784.373} C_VEL
LIN {X 0,Y 446.417,Z 370.877,A -85,B 0,C 180,E1 -8787.638,E2 -8787.638} C_VEL
LIN {X 0,Y 446.463,Z 370.869,A -85,B 0,C 180,E1 -8790.792,E2 -8790.792} C_VEL
LIN {X 0,Y 446.47,Z 370.868,A -85,B 0,C 180,E1 -8793.848,E2 -8793.848} C_VEL
LIN {X 0,Y 446.424,Z 370.875,A -85,B 0,C 180,E1 -8796.823,E2 -8796.823} C_VEL
LIN {X 0,Y 446.44,Z 370.872,A -85,B 0,C 180,E1 -8799.737,E2 -8799.737} C_VEL
LIN {X 0,Y 446.455,Z 370.87,A -85,B 0,C 180,E1 -8802.597,E2 -8802.597} C_VEL
LIN {X 0,Y 446.462,Z 370.872,A -85,B 0,C 180,E1 -8805.412,E2 -8805.412} C_VEL
LIN {X 0,Y 446.532,Z 370.859,A -85,B 0,C 180,E1 -8808.193,E2 -8808.193} C_VEL
LIN {X 0,Y 446.592,Z 370.851,A -85,B 0,C 180,E1 -8811.858,E2 -8811.858} C_VEL
LIN {X 0,Y 446.638,Z 370.848,A -85,B 0,C 180,E1 -8814.583,E2 -8814.583} C_VEL
LIN {X 0,Y 446.702,Z 370.841,A -85,B 0,C 180,E1 -8817.295,E2 -8817.295} C_VEL
LIN {X 0,Y 446.785,Z 370.827,A -85,B 0,C 180,E1 -8820,E2 -8820} C_VEL
LIN {X 0,Y 446.702,Z 370.843,A -85,B 0,C 180,E1 -8822.705,E2 -8822.705} C_VEL
LIN {X 0,Y 446.64,Z 370.847,A -85,B 0,C 180,E1 -8826.324,E2 -8826.324} C_VEL
LIN {X 0,Y 446.531,Z 370.863,A -85,B 0,C 180,E1 -8829.056,E2 -8829.056} C_VEL
LIN {X 0,Y 446.526,Z 370.867,A -85,B 0,C 180,E1 -8832.73,E2 -8832.73} C_VEL
LIN {X 0,Y 446.482,Z 370.869,A -85,B 0,C 180,E1 -8836.459,E2 -8836.459} C_VEL
LIN {X 0,Y 446.462,Z 370.868,A -85,B 0,C 180,E1 -8839.304,E2 -8839.304} C_VEL
LIN {X 0,Y 446.413,Z 370.876,A -85,B 0,C 180,E1 -8842.2,E2 -8842.2} C_VEL
LIN {X 0,Y 446.452,Z 370.87,A -85,B 0,C 180,E1 -8845.153,E2 -8845.153} C_VEL
LIN {X 0,Y 446.478,Z 370.868,A -85,B 0,C 180,E1 -8848.179,E2 -8848.179} C_VEL
LIN {X 0,Y 446.413,Z 370.874,A -85,B 0,C 180,E1 -8851.776,E2 -8851.776} C_VEL
LIN {X 0,Y 446.425,Z 370.879,A -85,B 0,C 180,E1 -8854.524,E2 -8854.524} C_VEL
LIN {X 0,Y 446.43,Z 370.875,A -85,B 0,C 180,E1 -8858.083,E2 -8858.083} C_VEL
LIN {X 0,Y 446.443,Z 370.871,A -85,B 0,C 180,E1 -8860.921,E2 -8860.921} C_VEL
LIN {X 0,Y 446.441,Z 370.872,A -85,B 0,C 180,E1 -8863.841,E2 -8863.841} C_VEL
LIN {X 0,Y 446.412,Z 370.88,A -85,B 0,C 180,E1 -8866.402,E2 -8866.402} C_VEL
LIN {X 0,Y 446.448,Z 370.871,A -85,B 0,C 180,E1 -8869.804,E2 -8869.804} C_VEL
LIN {X 0,Y 446.426,Z 370.878,A -85,B 0,C 180,E1 -8872.124,E2 -8872.124} C_VEL
LIN {X 0,Y 446.429,Z 370.872,A -85,B 0,C 180,E1 -8875.478,E2 -8875.478} C_VEL
LIN {X 0,Y 446.416,Z 370.875,A -85,B 0,C 180,E1 -8878.7,E2 -8878.7} C_VEL
LIN {X 0,Y 446.485,Z 370.869,A -85,B 0,C 180,E1 -8881.822,E2 -8881.822} C_VEL
LIN {X 0,Y 446.445,Z 370.874,A -85,B 0,C 180,E1 -8884.848,E2 -8884.848} C_VEL
LIN {X 0,Y 446.468,Z 370.961,A -85,B 0,C 180,E1 -8888.188,E2 -8888.188} C_VEL
LIN {X 0,Y 448.015,Z 379.392,A -85,B 0,C 180,E1 -8890.258,E2 -8890.258} C_VEL
LIN {X 0,Y 447.695,Z 387.98,A -85,B 0,C 180,E1 -8892.216,E2 -8892.216} C_VEL
LIN {X 0,Y 451.039,Z 404.911,A -85,B 0,C 180,E1 -8892.651,E2 -8892.651} C_VEL
LIN {X 0,Y 450.25,Z 495.162,A -85,B 0,C 180,E1 -8894.119,E2 -8894.119} C_VEL
LIN {X 0,Y 449.422,Z 500.942,A -85,B 0,C 180,E1 -8894.243,E2 -8894.243} C_VEL
LIN {X 0,Y 444.994,Z 513.872,A -85,B 0,C 180,E1 -8894.564,E2 -8894.564} C_VEL
LIN {X 0,Y 442.879,Z 521.198,A -85,B 0,C 180,E1 -8894.854,E2 -8894.854} C_VEL
LIN {X 0,Y 442.446,Z 524.752,A -85,B 0,C 180,E1 -8895.046,E2 -8895.046} C_VEL
LIN {X 0,Y 441.941,Z 536.174,A -85,B 0,C 180,E1 -8895.81,E2 -8895.81} C_VEL
LIN {X 0,Y 441.439,Z 546.474,A -85,B 0,C 180,E1 -8896.683,E2 -8896.683} C_VEL
LIN {X 0,Y 440.734,Z 557.067,A -85,B 0,C 180,E1 -8897.803,E2 -8897.803} C_VEL
LIN {X 0,Y 440.186,Z 565.9,A -85,B 0,C 180,E1 -8898.955,E2 -8898.955} C_VEL
LIN {X 0,Y 439.622,Z 574.517,A -85,B 0,C 180,E1 -8900.337,E2 -8900.337} C_VEL
LIN {X 0,Y 439.121,Z 581.386,A -85,B 0,C 180,E1 -8901.718,E2 -8901.718} C_VEL
LIN {X 0,Y 438.814,Z 587.266,A -85,B 0,C 180,E1 -8903.212,E2 -8903.212} C_VEL
LIN {X 0,Y 438.614,Z 591.195,A -85,B 0,C 180,E1 -8904.483,E2 -8904.483} C_VEL
LIN {X 0,Y 438.466,Z 593.479,A -85,B 0,C 180,E1 -8905.403,E2 -8905.403} C_VEL
LIN {X 0,Y 438.49,Z 595.332,A -85,B 0,C 180,E1 -8906.324,E2 -8906.324} C_VEL
LIN {X 0,Y 438.412,Z 596.732,A -85,B 0,C 180,E1 -8907.244,E2 -8907.244} C_VEL
LIN {X 0,Y 438.281,Z 598.343,A -85,B 0,C 180,E1 -8909.081,E2 -8909.081} C_VEL
LIN {X 0,Y 438.281,Z 598.577,A -85,B 0,C 180,E1 -8910,E2 -8910} C_VEL
LIN {X 0,Y 438.281,Z 598.39,A -85,B 0,C 180,E1 -8910.919,E2 -8910.919} C_VEL
LIN {X 0,Y 438.412,Z 596.842,A -85,B 0,C 180,E1 -8912.756,E2 -8912.756} C_VEL
LIN {X 0,Y 438.49,Z 595.489,A -85,B 0,C 180,E1 -8913.676,E2 -8913.676} C_VEL
LIN {X 0,Y 438.504,Z 592.635,A -85,B 0,C 180,E1 -8915.057,E2 -8915.057} C_VEL
LIN {X 0,Y 438.789,Z 588.755,A -85,B 0,C 180,E1 -8916.437,E2 -8916.437} C_VEL
LIN {X 0,Y 438.997,Z 583.755,A -85,B 0,C 180,E1 -8917.821,E2 -8917.821} C_VEL
LIN {X 0,Y 439.405,Z 577.457,A -85,B 0,C 180,E1 -8919.203,E2 -8919.203} C_VEL
LIN {X 0,Y 439.88,Z 569.571,A -85,B 0,C 180,E1 -8920.587,E2 -8920.587} C_VEL
LIN {X 0,Y 440.385,Z 561.53,A -85,B 0,C 180,E1 -8921.74,E2 -8921.74} C_VEL
LIN {X 0,Y 441.117,Z 551.708,A -85,B 0,C 180,E1 -8922.888,E2 -8922.888} C_VEL
LIN {X 0,Y 441.67,Z 540.816,A -85,B 0,C 180,E1 -8923.914,E2 -8923.914} C_VEL
LIN {X 0,Y 442.282,Z 529.841,A -85,B 0,C 180,E1 -8924.728,E2 -8924.728} C_VEL
LIN {X 0,Y 442.75,Z 517.881,A -85,B 0,C 180,E1 -8925.419,E2 -8925.419} C_VEL
LIN {X 0,Y 443.245,Z 504.75,A -85,B 0,C 180,E1 -8925.962,E2 -8925.962} C_VEL
LIN {X 0,Y 443.483,Z 491.539,A -85,B 0,C 180,E1 -8926.307,E2 -8926.307} C_VEL
LIN {X 0,Y 444.291,Z 405.519,A -85,B 0,C 180,E1 -8927.71,E2 -8927.71} C_VEL
LIN {X 0,Y 440.775,Z 388.275,A -85,B 0,C 180,E1 -8928.163,E2 -8928.163} C_VEL
LIN {X 0,Y 441.078,Z 380.599,A -85,B 0,C 180,E1 -8929.933,E2 -8929.933} C_VEL
LIN {X 0,Y 439.372,Z 371.763,A -85,B 0,C 180,E1 -8932.154,E2 -8932.154} C_VEL
LIN {X 0,Y 439.417,Z 371.753,A -85,B 0,C 180,E1 -8934.572,E2 -8934.572} C_VEL
LIN {X 0,Y 439.441,Z 371.745,A -85,B 0,C 180,E1 -8937.632,E2 -8937.632} C_VEL
LIN {X 0,Y 439.361,Z 371.752,A -85,B 0,C 180,E1 -8940.788,E2 -8940.788} C_VEL
LIN {X 0,Y 439.387,Z 371.755,A -85,B 0,C 180,E1 -8944.043,E2 -8944.043} C_VEL
LIN {X 0,Y 439.355,Z 371.753,A -85,B 0,C 180,E1 -8946.888,E2 -8946.888} C_VEL
LIN {X 0,Y 439.411,Z 371.753,A -85,B 0,C 180,E1 -8949.85,E2 -8949.85} C_VEL
LIN {X 0,Y 439.379,Z 371.75,A -85,B 0,C 180,E1 -8952.626,E2 -8952.626} C_VEL
LIN {X 0,Y 439.399,Z 371.751,A -85,B 0,C 180,E1 -8956.033,E2 -8956.033} C_VEL
LIN {X 0,Y 439.396,Z 371.748,A -85,B 0,C 180,E1 -8959.021,E2 -8959.021} C_VEL
LIN {X 0,Y 439.385,Z 371.756,A -85,B 0,C 180,E1 -8961.604,E2 -8961.604} C_VEL
LIN {X 0,Y 439.396,Z 371.748,A -85,B 0,C 180,E1 -8964.843,E2 -8964.843} C_VEL
LIN {X 0,Y 439.369,Z 371.752,A -85,B 0,C 180,E1 -8968.139,E2 -8968.139} C_VEL
LIN {X 0,Y 439.426,Z 371.751,A -85,B 0,C 180,E1 -8971.597,E2 -8971.597} C_VEL
LIN {X 0,Y 439.398,Z 371.747,A -85,B 0,C 180,E1 -8974.415,E2 -8974.415} C_VEL
LIN {X 0,Y 439.36,Z 371.76,A -85,B 0,C 180,E1 -8977.424,E2 -8977.424} C_VEL
LIN {X 0,Y 439.434,Z 371.743,A -85,B 0,C 180,E1 -8980.662,E2 -8980.662} C_VEL
LIN {X 0,Y 439.455,Z 371.74,A -85,B 0,C 180,E1 -8984.224,E2 -8984.224} C_VEL
LIN {X 0,Y 439.5,Z 371.735,A -85,B 0,C 180,E1 -8988.002,E2 -8988.002} C_VEL
LIN {X 0,Y 439.539,Z 371.732,A -85,B 0,C 180,E1 -8991.726,E2 -8991.726} C_VEL
LIN {X 0,Y 439.613,Z 371.721,A -85,B 0,C 180,E1 -8994.496,E2 -8994.496} C_VEL
LIN {X 0,Y 439.628,Z 371.719,A -85,B 0,C 180,E1 -8998.168,E2 -8998.168} C_VEL
LIN {X 0,Y 439.756,Z 371.703,A -85,B 0,C 180,E1 -9000,E2 -9000} C_VEL
LIN {X 0,Y 439.65,Z 371.72,A -85,B 0,C 180,E1 -9002.749,E2 -9002.749} C_VEL
LIN {X 0,Y 439.611,Z 371.722,A -85,B 0,C 180,E1 -9006.425,E2 -9006.425} C_VEL
LIN {X 0,Y 439.494,Z 371.74,A -85,B 0,C 180,E1 -9009.202,E2 -9009.202} C_VEL
LIN {X 0,Y 439.495,Z 371.74,A -85,B 0,C 180,E1 -9012.727,E2 -9012.727} C_VEL
LIN {X 0,Y 439.439,Z 371.744,A -85,B 0,C 180,E1 -9016.349,E2 -9016.349} C_VEL
LIN {X 0,Y 439.396,Z 371.748,A -85,B 0,C 180,E1 -9019.627,E2 -9019.627} C_VEL
LIN {X 0,Y 439.359,Z 371.757,A -85,B 0,C 180,E1 -9022.576,E2 -9022.576} C_VEL
LIN {X 0,Y 439.398,Z 371.747,A -85,B 0,C 180,E1 -9025.585,E2 -9025.585} C_VEL
LIN {X 0,Y 439.41,Z 371.753,A -85,B 0,C 180,E1 -9028.674,E2 -9028.674} C_VEL
LIN {X 0,Y 439.364,Z 371.753,A -85,B 0,C 180,E1 -9032.031,E2 -9032.031} C_VEL
LIN {X 0,Y 439.39,Z 371.749,A -85,B 0,C 180,E1 -9035.341,E2 -9035.341} C_VEL
LIN {X 0,Y 439.393,Z 371.755,A -85,B 0,C 180,E1 -9038.594,E2 -9038.594} C_VEL
LIN {X 0,Y 439.4,Z 371.748,A -85,B 0,C 180,E1 -9041.26,E2 -9041.26} C_VEL
LIN {X 0,Y 439.406,Z 371.751,A -85,B 0,C 180,E1 -9044.729,E2 -9044.729} C_VEL
LIN {X 0,Y 439.394,Z 371.749,A -85,B 0,C 180,E1 -9047.797,E2 -9047.797} C_VEL
LIN {X 0,Y 439.434,Z 371.748,A -85,B 0,C 180,E1 -9050.229,E2 -9050.229} C_VEL
LIN {X 0,Y 439.375,Z 371.751,A -85,B 0,C 180,E1 -9053.714,E2 -9053.714} C_VEL
LIN {X 0,Y 439.374,Z 371.751,A -85,B 0,C 180,E1 -9057.055,E2 -9057.055} C_VEL
LIN {X 0,Y 439.382,Z 371.757,A -85,B 0,C 180,E1 -9060.275,E2 -9060.275} C_VEL
LIN {X 0,Y 439.495,Z 371.847,A -85,B 0,C 180,E1 -9062.856,E2 -9062.856} C_VEL
LIN {X 0,Y 442.128,Z 385.128,A -85,B 0,C 180,E1 -9065.589,E2 -9065.589} C_VEL
LIN {X 0,Y 441.96,Z 392.621,A -85,B 0,C 180,E1 -9067.012,E2 -9067.012} C_VEL
LIN {X 0,Y 440.835,Z 412.361,A -85,B 0,C 180,E1 -9070.683,E2 -9070.683} C_VEL
LIN {X 0,Y 440.481,Z 418.722,A -85,B 0,C 180,E1 -9071.864,E2 -9071.864} C_VEL
LIN {X 0,Y 444.042,Z 442.114,A -85,B 0,C 180,E1 -9072.404,E2 -9072.404} C_VEL
LIN {X 0,Y 443.225,Z 527.103,A -85,B 0,C 180,E1 -9073.801,E2 -9073.801} C_VEL
LIN {X 0,Y 442.808,Z 540.363,A -85,B 0,C 180,E1 -9074.2,E2 -9074.2} C_VEL
LIN {X 0,Y 442.186,Z 553.644,A -85,B 0,C 180,E1 -9074.797,E2 -9074.797} C_VEL
LIN {X 0,Y 441.599,Z 564.797,A -85,B 0,C 180,E1 -9075.484,E2 -9075.484} C_VEL
LIN {X 0,Y 440.936,Z 575.501,A -85,B 0,C 180,E1 -9076.321,E2 -9076.321} C_VEL
LIN {X 0,Y 440.302,Z 586.858,A -85,B 0,C 180,E1 -9077.439,E2 -9077.439} C_VEL
LIN {X 0,Y 439.847,Z 595.41,A -85,B 0,C 180,E1 -9078.479,E2 -9078.479} C_VEL
LIN {X 0,Y 439.304,Z 603.299,A -85,B 0,C 180,E1 -9079.632,E2 -9079.632} C_VEL
LIN {X 0,Y 438.879,Z 611.009,A -85,B 0,C 180,E1 -9081.018,E2 -9081.018} C_VEL
LIN {X 0,Y 438.553,Z 618.121,A -85,B 0,C 180,E1 -9082.634,E2 -9082.634} C_VEL
LIN {X 0,Y 438.37,Z 622.781,A -85,B 0,C 180,E1 -9083.995,E2 -9083.995} C_VEL
LIN {X 0,Y 438.342,Z 626.473,A -85,B 0,C 180,E1 -9085.402,E2 -9085.402} C_VEL
LIN {X 0,Y 438.283,Z 628.338,A -85,B 0,C 180,E1 -9086.323,E2 -9086.323} C_VEL
LIN {X 0,Y 438.341,Z 629.74,A -85,B 0,C 180,E1 -9087.243,E2 -9087.243} C_VEL
LIN {X 0,Y 438.277,Z 631.347,A -85,B 0,C 180,E1 -9089.081,E2 -9089.081} C_VEL
LIN {X 0,Y 438.28,Z 631.564,A -85,B 0,C 180,E1 -9090,E2 -9090} C_VEL
LIN {X 0,Y 438.277,Z 631.346,A -85,B 0,C 180,E1 -9090.919,E2 -9090.919} C_VEL
LIN {X 0,Y 438.341,Z 629.741,A -85,B 0,C 180,E1 -9092.757,E2 -9092.757} C_VEL
LIN {X 0,Y 438.283,Z 628.337,A -85,B 0,C 180,E1 -9093.677,E2 -9093.677} C_VEL
LIN {X 0,Y 438.384,Z 625.395,A -85,B 0,C 180,E1 -9095.058,E2 -9095.058} C_VEL
LIN {X 0,Y 438.448,Z 621.409,A -85,B 0,C 180,E1 -9096.442,E2 -9096.442} C_VEL
LIN {X 0,Y 438.682,Z 615.284,A -85,B 0,C 180,E1 -9098.058,E2 -9098.058} C_VEL
LIN {X 0,Y 439.013,Z 608.593,A -85,B 0,C 180,E1 -9099.444,E2 -9099.444} C_VEL
LIN {X 0,Y 439.472,Z 600.294,A -85,B 0,C 180,E1 -9100.83,E2 -9100.83} C_VEL
LIN {X 0,Y 440.057,Z 591.794,A -85,B 0,C 180,E1 -9101.983,E2 -9101.983} C_VEL
LIN {X 0,Y 440.61,Z 581.929,A -85,B 0,C 180,E1 -9103.074,E2 -9103.074} C_VEL
LIN {X 0,Y 441.241,Z 570.901,A -85,B 0,C 180,E1 -9104.057,E2 -9104.057} C_VEL
LIN {X 0,Y 441.867,Z 559.516,A -85,B 0,C 180,E1 -9104.86,E2 -9104.86} C_VEL
LIN {X 0,Y 442.478,Z 547.838,A -85,B 0,C 180,E1 -9105.488,E2 -9105.488} C_VEL
LIN {X 0,Y 442.935,Z 536.214,A -85,B 0,C 180,E1 -9105.943,E2 -9105.943} C_VEL
LIN {X 0,Y 443.296,Z 522.595,A -85,B 0,C 180,E1 -9106.285,E2 -9106.285} C_VEL
LIN {X 0,Y 443.962,Z 441.043,A -85,B 0,C 180,E1 -9107.613,E2 -9107.613} C_VEL
LIN {X 0,Y 440.494,Z 418.64,A -85,B 0,C 180,E1 -9108.148,E2 -9108.148} C_VEL
LIN {X 0,Y 441.52,Z 399.388,A -85,B 0,C 180,E1 -9111.72,E2 -9111.72} C_VEL
LIN {X 0,Y 442.261,Z 386.403,A -85,B 0,C 180,E1 -9114.154,E2 -9114.154} C_VEL
LIN {X 0,Y 440.039,Z 374.567,A -85,B 0,C 180,E1 -9116.569,E2 -9116.569} C_VEL
LIN {X 0,Y 439.471,Z 371.745,A -85,B 0,C 180,E1 -9117.178,E2 -9117.178} C_VEL
LIN {X 0,Y 439.38,Z 371.756,A -85,B 0,C 180,E1 -9120.26,E2 -9120.26} C_VEL
LIN {X 0,Y 439.395,Z 371.755,A -85,B 0,C 180,E1 -9123.723,E2 -9123.723} C_VEL
LIN {X 0,Y 439.355,Z 371.753,A -85,B 0,C 180,E1 -9126.888,E2 -9126.888} C_VEL
LIN {X 0,Y 439.41,Z 371.751,A -85,B 0,C 180,E1 -9129.85,E2 -9129.85} C_VEL
LIN {X 0,Y 439.382,Z 371.749,A -85,B 0,C 180,E1 -9132.627,E2 -9132.627} C_VEL
LIN {X 0,Y 439.399,Z 371.749,A -85,B 0,C 180,E1 -9136.033,E2 -9136.033} C_VEL
LIN {X 0,Y 439.396,Z 371.75,A -85,B 0,C 180,E1 -9139.021,E2 -9139.021} C_VEL
LIN {X 0,Y 439.386,Z 371.755,A -85,B 0,C 180,E1 -9141.604,E2 -9141.604} C_VEL
LIN {X 0,Y 439.395,Z 371.749,A -85,B 0,C 180,E1 -9144.844,E2 -9144.844} C_VEL
LIN {X 0,Y 439.368,Z 371.751,A -85,B 0,C 180,E1 -9148.139,E2 -9148.139} C_VEL
LIN {X 0,Y 439.418,Z 371.753,A -85,B 0,C 180,E1 -9151.327,E2 -9151.327} C_VEL
LIN {X 0,Y 439.398,Z 371.747,A -85,B 0,C 180,E1 -9154.415,E2 -9154.415} C_VEL
LIN {X 0,Y 439.359,Z 371.758,A -85,B 0,C 180,E1 -9157.424,E2 -9157.424} C_VEL
LIN {X 0,Y 439.433,Z 371.745,A -85,B 0,C 180,E1 -9160.662,E2 -9160.662} C_VEL
LIN {X 0,Y 439.454,Z 371.74,A -85,B 0,C 180,E1 -9164.224,E2 -9164.224} C_VEL
LIN {X 0,Y 439.5,Z 371.735,A -85,B 0,C 180,E1 -9168.002,E2 -9168.002} C_VEL
LIN {X 0,Y 439.539,Z 371.73,A -85,B 0,C 180,E1 -9171.726,E2 -9171.726} C_VEL
LIN {X 0,Y 439.613,Z 371.722,A -85,B 0,C 180,E1 -9174.496,E2 -9174.496} C_VEL
LIN {X 0,Y 439.628,Z 371.719,A -85,B 0,C 180,E1 -9178.168,E2 -9178.168} C_VEL
LIN {X 0,Y 439.756,Z 371.703,A -85,B 0,C 180,E1 -9180,E2 -9180} C_VEL
LIN {X 0,Y 439.649,Z 371.722,A -85,B 0,C 180,E1 -9182.749,E2 -9182.749} C_VEL
LIN {X 0,Y 439.611,Z 371.723,A -85,B 0,C 180,E1 -9186.425,E2 -9186.425} C_VEL
LIN {X 0,Y 439.493,Z 371.738,A -85,B 0,C 180,E1 -9189.202,E2 -9189.202} C_VEL
LIN {X 0,Y 439.496,Z 371.743,A -85,B 0,C 180,E1 -9192.727,E2 -9192.727} C_VEL
LIN {X 0,Y 439.439,Z 371.745,A -85,B 0,C 180,E1 -9196.349,E2 -9196.349} C_VEL
LIN {X 0,Y 439.396,Z 371.748,A -85,B 0,C 180,E1 -9199.627,E2 -9199.627} C_VEL
LIN {X 0,Y 439.36,Z 371.759,A -85,B 0,C 180,E1 -9202.576,E2 -9202.576} C_VEL
LIN {X 0,Y 439.398,Z 371.747,A -85,B 0,C 180,E1 -9205.585,E2 -9205.585} C_VEL
LIN {X 0,Y 439.411,Z 371.752,A -85,B 0,C 180,E1 -9208.674,E2 -9208.674} C_VEL
LIN {X 0,Y 439.364,Z 371.754,A -85,B 0,C 180,E1 -9212.031,E2 -9212.031} C_VEL
LIN {X 0,Y 439.39,Z 371.748,A -85,B 0,C 180,E1 -9215.341,E2 -9215.341} C_VEL
LIN {X 0,Y 439.391,Z 371.754,A -85,B 0,C 180,E1 -9218.594,E2 -9218.594} C_VEL
LIN {X 0,Y 439.401,Z 371.747,A -85,B 0,C 180,E1 -9221.26,E2 -9221.26} C_VEL
LIN {X 0,Y 439.405,Z 371.749,A -85,B 0,C 180,E1 -9224.729,E2 -9224.729} C_VEL
LIN {X 0,Y 439.393,Z 371.75,A -85,B 0,C 180,E1 -9227.797,E2 -9227.797} C_VEL
LIN {X 0,Y 439.434,Z 371.75,A -85,B 0,C 180,E1 -9230.229,E2 -9230.229} C_VEL
LIN {X 0,Y 439.376,Z 371.752,A -85,B 0,C 180,E1 -9233.714,E2 -9233.714} C_VEL
LIN {X 0,Y 439.371,Z 371.751,A -85,B 0,C 180,E1 -9237.055,E2 -9237.055} C_VEL
LIN {X 0,Y 439.383,Z 371.755,A -85,B 0,C 180,E1 -9240.275,E2 -9240.275} C_VEL
LIN {X 0,Y 439.429,Z 371.744,A -85,B 0,C 180,E1 -9243.397,E2 -9243.397} C_VEL
LIN {X 0,Y 439.385,Z 371.757,A -85,B 0,C 180,E1 -9246.43,E2 -9246.43} C_VEL
LIN {X 0,Y 439.417,Z 371.894,A -85,B 0,C 180,E1 -9247.991,E2 -9247.991} C_VEL
LIN {X 0,Y 441.005,Z 380.324,A -85,B 0,C 180,E1 -9250.093,E2 -9250.093} C_VEL
LIN {X 0,Y 440.776,Z 388.295,A -85,B 0,C 180,E1 -9251.939,E2 -9251.939} C_VEL
LIN {X 0,Y 444.284,Z 405.743,A -85,B 0,C 180,E1 -9252.388,E2 -9252.388} C_VEL
LIN {X 0,Y 443.451,Z 495.459,A -85,B 0,C 180,E1 -9253.869,E2 -9253.869} C_VEL
LIN {X 0,Y 443.022,Z 509.304,A -85,B 0,C 180,E1 -9254.296,E2 -9254.296} C_VEL
LIN {X 0,Y 442.57,Z 521.693,A -85,B 0,C 180,E1 -9254.869,E2 -9254.869} C_VEL
LIN {X 0,Y 442.446,Z 524.752,A -85,B 0,C 180,E1 -9255.046,E2 -9255.046} C_VEL
LIN {X 0,Y 441.6,Z 530.1,A -85,B 0,C 180,E1 -9255.354,E2 -9255.354} C_VEL
LIN {X 0,Y 438.493,Z 538.634,A -85,B 0,C 180,E1 -9255.871,E2 -9255.871} C_VEL
LIN {X 0,Y 435.25,Z 546.744,A -85,B 0,C 180,E1 -9256.484,E2 -9256.484} C_VEL
LIN {X 0,Y 434.204,Z 551.427,A -85,B 0,C 180,E1 -9256.937,E2 -9256.937} C_VEL
LIN {X 0,Y 433.494,Z 561.09,A -85,B 0,C 180,E1 -9258.071,E2 -9258.071} C_VEL
LIN {X 0,Y 432.957,Z 569.248,A -85,B 0,C 180,E1 -9259.241,E2 -9259.241} C_VEL
LIN {X 0,Y 432.399,Z 577.238,A -85,B 0,C 180,E1 -9260.646,E2 -9260.646} C_VEL
LIN {X 0,Y 431.984,Z 583.65,A -85,B 0,C 180,E1 -9262.051,E2 -9262.051} C_VEL
LIN {X 0,Y 431.731,Z 588.735,A -85,B 0,C 180,E1 -9263.457,E2 -9263.457} C_VEL
LIN {X 0,Y 431.449,Z 592.687,A -85,B 0,C 180,E1 -9264.86,E2 -9264.86} C_VEL
LIN {X 0,Y 431.397,Z 595.6,A -85,B 0,C 180,E1 -9266.264,E2 -9266.264} C_VEL
LIN {X 0,Y 431.345,Z 596.999,A -85,B 0,C 180,E1 -9267.198,E2 -9267.198} C_VEL
LIN {X 0,Y 431.196,Z 598.61,A -85,B 0,C 180,E1 -9269.066,E2 -9269.066} C_VEL
LIN {X 0,Y 431.194,Z 598.844,A -85,B 0,C 180,E1 -9270,E2 -9270} C_VEL
LIN {X 0,Y 431.196,Z 598.657,A -85,B 0,C 180,E1 -9270.934,E2 -9270.934} C_VEL
LIN {X 0,Y 431.345,Z 597.107,A -85,B 0,C 180,E1 -9272.802,E2 -9272.802} C_VEL
LIN {X 0,Y 431.396,Z 595.756,A -85,B 0,C 180,E1 -9273.736,E2 -9273.736} C_VEL
LIN {X 0,Y 431.447,Z 592.901,A -85,B 0,C 180,E1 -9275.14,E2 -9275.14} C_VEL
LIN {X 0,Y 431.72,Z 589.021,A -85,B 0,C 180,E1 -9276.543,E2 -9276.543} C_VEL
LIN {X 0,Y 431.948,Z 584.021,A -85,B 0,C 180,E1 -9277.949,E2 -9277.949} C_VEL
LIN {X 0,Y 432.382,Z 577.722,A -85,B 0,C 180,E1 -9279.354,E2 -9279.354} C_VEL
LIN {X 0,Y 432.906,Z 569.835,A -85,B 0,C 180,E1 -9280.76,E2 -9280.76} C_VEL
LIN {X 0,Y 433.431,Z 561.793,A -85,B 0,C 180,E1 -9281.931,E2 -9281.931} C_VEL
LIN {X 0,Y 434.21,Z 551.971,A -85,B 0,C 180,E1 -9283.097,E2 -9283.097} C_VEL
LIN {X 0,Y 434.801,Z 541.077,A -85,B 0,C 180,E1 -9284.138,E2 -9284.138} C_VEL
LIN {X 0,Y 435.422,Z 530.101,A -85,B 0,C 180,E1 -9284.966,E2 -9284.966} C_VEL
LIN {X 0,Y 435.938,Z 518.139,A -85,B 0,C 180,E1 -9285.666,E2 -9285.666} C_VEL
LIN {X 0,Y 436.434,Z 505.003,A -85,B 0,C 180,E1 -9286.217,E2 -9286.217} C_VEL
LIN {X 0,Y 436.691,Z 491.783,A -85,B 0,C 180,E1 -9286.568,E2 -9286.568} C_VEL
LIN {X 0,Y 437.502,Z 406.327,A -85,B 0,C 180,E1 -9287.984,E2 -9287.984} C_VEL
LIN {X 0,Y 433.883,Z 388.557,A -85,B 0,C 180,E1 -9288.455,E2 -9288.455} C_VEL
LIN {X 0,Y 434.06,Z 381.56,A -85,B 0,C 180,E1 -9290.099,E2 -9290.099} C_VEL
LIN {X 0,Y 432.326,Z 372.641,A -85,B 0,C 180,E1 -9292.363,E2 -9292.363} C_VEL
LIN {X 0,Y 432.353,Z 372.631,A -85,B 0,C 180,E1 -9295.001,E2 -9295.001} C_VEL
LIN {X 0,Y 432.382,Z 372.627,A -85,B 0,C 180,E1 -9298.123,E2 -9298.123} C_VEL
LIN {X 0,Y 432.321,Z 372.63,A -85,B 0,C 180,E1 -9301.345,E2 -9301.345} C_VEL
LIN {X 0,Y 432.34,Z 372.627,A -85,B 0,C 180,E1 -9304.676,E2 -9304.676} C_VEL
LIN {X 0,Y 432.346,Z 372.63,A -85,B 0,C 180,E1 -9308.148,E2 -9308.148} C_VEL
LIN {X 0,Y 432.33,Z 372.633,A -85,B 0,C 180,E1 -9311.601,E2 -9311.601} C_VEL
LIN {X 0,Y 432.334,Z 372.629,A -85,B 0,C 180,E1 -9314.346,E2 -9314.346} C_VEL
LIN {X 0,Y 432.362,Z 372.624,A -85,B 0,C 180,E1 -9317.008,E2 -9317.008} C_VEL
LIN {X 0,Y 432.353,Z 372.631,A -85,B 0,C 180,E1 -9319.816,E2 -9319.816} C_VEL
LIN {X 0,Y 432.311,Z 372.631,A -85,B 0,C 180,E1 -9323.022,E2 -9323.022} C_VEL
LIN {X 0,Y 432.354,Z 372.628,A -85,B 0,C 180,E1 -9325.996,E2 -9325.996} C_VEL
LIN {X 0,Y 432.341,Z 372.634,A -85,B 0,C 180,E1 -9329.489,E2 -9329.489} C_VEL
LIN {X 0,Y 432.386,Z 372.622,A -85,B 0,C 180,E1 -9332.928,E2 -9332.928} C_VEL
LIN {X 0,Y 432.365,Z 372.625,A -85,B 0,C 180,E1 -9336.023,E2 -9336.023} C_VEL
LIN {X 0,Y 432.347,Z 372.629,A -85,B 0,C 180,E1 -9339.046,E2 -9339.046} C_VEL
LIN {X 0,Y 432.37,Z 372.624,A -85,B 0,C 180,E1 -9342.011,E2 -9342.011} C_VEL
LIN {X 0,Y 432.388,Z 372.623,A -85,B 0,C 180,E1 -9344.926,E2 -9344.926} C_VEL
LIN {X 0,Y 432.473,Z 372.612,A -85,B 0,C 180,E1 -9347.804,E2 -9347.804} C_VEL
LIN {X 0,Y 432.484,Z 372.612,A -85,B 0,C 180,E1 -9351.59,E2 -9351.59} C_VEL
LIN {X 0,Y 432.59,Z 372.596,A -85,B 0,C 180,E1 -9354.406,E2 -9354.406} C_VEL
LIN {X 0,Y 432.598,Z 372.594,A -85,B 0,C 180,E1 -9358.138,E2 -9358.138} C_VEL
LIN {X 0,Y 432.726,Z 372.578,A -85,B 0,C 180,E1 -9360,E2 -9360} C_VEL
LIN {X 0,Y 432.599,Z 372.598,A -85,B 0,C 180,E1 -9362.794,E2 -9362.794} C_VEL
LIN {X 0,Y 432.566,Z 372.601,A -85,B 0,C 180,E1 -9366.53,E2 -9366.53} C_VEL
LIN {X 0,Y 432.437,Z 372.617,A -85,B 0,C 180,E1 -9369.353,E2 -9369.353} C_VEL
LIN {X 0,Y 432.436,Z 372.621,A -85,B 0,C 180,E1 -9372.812,E2 -9372.812} C_VEL
LIN {X 0,Y 432.404,Z 372.621,A -85,B 0,C 180,E1 -9376.479,E2 -9376.479} C_VEL
LIN {X 0,Y 432.333,Z 372.628,A -85,B 0,C 180,E1 -9379.961,E2 -9379.961} C_VEL
LIN {X 0,Y 432.313,Z 372.635,A -85,B 0,C 180,E1 -9382.965,E2 -9382.965} C_VEL
LIN {X 0,Y 432.358,Z 372.625,A -85,B 0,C 180,E1 -9386.033,E2 -9386.033} C_VEL
LIN {X 0,Y 432.336,Z 372.629,A -85,B 0,C 180,E1 -9389.188,E2 -9389.188} C_VEL
LIN {X 0,Y 432.317,Z 372.634,A -85,B 0,C 180,E1 -9392.444,E2 -9392.444} C_VEL
LIN {X 0,Y 432.34,Z 372.626,A -85,B 0,C 180,E1 -9395.633,E2 -9395.633} C_VEL
LIN {X 0,Y 432.362,Z 372.624,A -85,B 0,C 180,E1 -9399.342,E2 -9399.342} C_VEL
LIN {X 0,Y 432.369,Z 372.623,A -85,B 0,C 180,E1 -9401.793,E2 -9401.793} C_VEL
LIN {X 0,Y 432.374,Z 372.628,A -85,B 0,C 180,E1 -9404.342,E2 -9404.342} C_VEL
LIN {X 0,Y 432.332,Z 372.632,A -85,B 0,C 180,E1 -9408.204,E2 -9408.204} C_VEL
LIN {X 0,Y 432.35,Z 372.625,A -85,B 0,C 180,E1 -9411.284,E2 -9411.284} C_VEL
LIN {X 0,Y 432.344,Z 372.633,A -85,B 0,C 180,E1 -9414.369,E2 -9414.369} C_VEL
LIN {X 0,Y 432.326,Z 372.629,A -85,B 0,C 180,E1 -9417.558,E2 -9417.558} C_VEL
LIN {X 0,Y 432.343,Z 372.63,A -85,B 0,C 180,E1 -9420.813,E2 -9420.813} C_VEL
LIN {X 0,Y 432.457,Z 372.751,A -85,B 0,C 180,E1 -9422.606,E2 -9422.606} C_VEL
LIN {X 0,Y 435.126,Z 386.188,A -85,B 0,C 180,E1 -9425.424,E2 -9425.424} C_VEL
LIN {X 0,Y 435.204,Z 391.522,A -85,B 0,C 180,E1 -9426.468,E2 -9426.468} C_VEL
LIN {X 0,Y 433.959,Z 410.81,A -85,B 0,C 180,E1 -9430.118,E2 -9430.118} C_VEL
LIN {X 0,Y 433.547,Z 418.46,A -85,B 0,C 180,E1 -9431.565,E2 -9431.565} C_VEL
LIN {X 0,Y 437.259,Z 442.628,A -85,B 0,C 180,E1 -9432.135,E2 -9432.135} C_VEL
LIN {X 0,Y 436.416,Z 526.848,A -85,B 0,C 180,E1 -9433.541,E2 -9433.541} C_VEL
LIN {X 0,Y 435.975,Z 540.103,A -85,B 0,C 180,E1 -9433.945,E2 -9433.945} C_VEL
LIN {X 0,Y 435.319,Z 553.381,A -85,B 0,C 180,E1 -9434.551,E2 -9434.551} C_VEL
LIN {X 0,Y 434.715,Z 564.533,A -85,B 0,C 180,E1 -9435.249,E2 -9435.249} C_VEL
LIN {X 0,Y 433.938,Z 576.341,A -85,B 0,C 180,E1 -9436.198,E2 -9436.198} C_VEL
LIN {X 0,Y 433.35,Z 586.592,A -85,B 0,C 180,E1 -9437.234,E2 -9437.234} C_VEL
LIN {X 0,Y 432.855,Z 595.144,A -85,B 0,C 180,E1 -9438.29,E2 -9438.29} C_VEL
LIN {X 0,Y 432.268,Z 603.032,A -85,B 0,C 180,E1 -9439.461,E2 -9439.461} C_VEL
LIN {X 0,Y 431.831,Z 610.742,A -85,B 0,C 180,E1 -9440.87,E2 -9440.87} C_VEL
LIN {X 0,Y 431.498,Z 617.854,A -85,B 0,C 180,E1 -9442.513,E2 -9442.513} C_VEL
LIN {X 0,Y 431.27,Z 622.944,A -85,B 0,C 180,E1 -9444.037,E2 -9444.037} C_VEL
LIN {X 0,Y 431.271,Z 626.206,A -85,B 0,C 180,E1 -9445.326,E2 -9445.326} C_VEL
LIN {X 0,Y 431.19,Z 628.071,A -85,B 0,C 180,E1 -9446.262,E2 -9446.262} C_VEL
LIN {X 0,Y 431.237,Z 629.473,A -85,B 0,C 180,E1 -9447.198,E2 -9447.198} C_VEL
LIN {X 0,Y 431.218,Z 630.472,A -85,B 0,C 180,E1 -9448.132,E2 -9448.132} C_VEL
LIN {X 0,Y 431.193,Z 631.08,A -85,B 0,C 180,E1 -9449.066,E2 -9449.066} C_VEL
LIN {X 0,Y 431.192,Z 631.297,A -85,B 0,C 180,E1 -9450,E2 -9450} C_VEL
LIN {X 0,Y 431.193,Z 631.079,A -85,B 0,C 180,E1 -9450.934,E2 -9450.934} C_VEL
LIN {X 0,Y 431.218,Z 630.471,A -85,B 0,C 180,E1 -9451.868,E2 -9451.868} C_VEL
LIN {X 0,Y 431.237,Z 629.473,A -85,B 0,C 180,E1 -9452.802,E2 -9452.802} C_VEL
LIN {X 0,Y 431.19,Z 628.069,A -85,B 0,C 180,E1 -9453.738,E2 -9453.738} C_VEL
LIN {X 0,Y 431.294,Z 625.127,A -85,B 0,C 180,E1 -9455.142,E2 -9455.142} C_VEL
LIN {X 0,Y 431.376,Z 621.14,A -85,B 0,C 180,E1 -9456.548,E2 -9456.548} C_VEL
LIN {X 0,Y 431.615,Z 615.014,A -85,B 0,C 180,E1 -9458.191,E2 -9458.191} C_VEL
LIN {X 0,Y 431.972,Z 608.323,A -85,B 0,C 180,E1 -9459.599,E2 -9459.599} C_VEL
LIN {X 0,Y 432.45,Z 600.023,A -85,B 0,C 180,E1 -9461.008,E2 -9461.008} C_VEL
LIN {X 0,Y 433.077,Z 591.523,A -85,B 0,C 180,E1 -9462.179,E2 -9462.179} C_VEL
LIN {X 0,Y 433.639,Z 582.121,A -85,B 0,C 180,E1 -9463.241,E2 -9463.241} C_VEL
LIN {X 0,Y 434.326,Z 570.629,A -85,B 0,C 180,E1 -9464.286,E2 -9464.286} C_VEL
LIN {X 0,Y 434.988,Z 559.243,A -85,B 0,C 180,E1 -9465.101,E2 -9465.101} C_VEL
LIN {X 0,Y 435.625,Z 547.564,A -85,B 0,C 180,E1 -9465.738,E2 -9465.738} C_VEL
LIN {X 0,Y 436.148,Z 535.022,A -85,B 0,C 180,E1 -9466.228,E2 -9466.228} C_VEL
LIN {X 0,Y 436.482,Z 522.313,A -85,B 0,C 180,E1 -9466.546,E2 -9466.546} C_VEL
LIN {X 0,Y 437.207,Z 441.934,A -85,B 0,C 180,E1 -9467.875,E2 -9467.875} C_VEL
LIN {X 0,Y 433.538,Z 418.445,A -85,B 0,C 180,E1 -9468.436,E2 -9468.436} C_VEL
LIN {X 0,Y 434.575,Z 400.432,A -85,B 0,C 180,E1 -9471.836,E2 -9471.836} C_VEL
LIN {X 0,Y 435.312,Z 387.464,A -85,B 0,C 180,E1 -9474.31,E2 -9474.31} C_VEL
LIN {X 0,Y 432.78,Z 374.351,A -85,B 0,C 180,E1 -9477.045,E2 -9477.045} C_VEL
LIN {X 0,Y 432.422,Z 372.622,A -85,B 0,C 180,E1 -9477.462,E2 -9477.462} C_VEL
LIN {X 0,Y 432.347,Z 372.631,A -85,B 0,C 180,E1 -9480.51,E2 -9480.51} C_VEL
LIN {X 0,Y 432.358,Z 372.628,A -85,B 0,C 180,E1 -9484.003,E2 -9484.003} C_VEL
LIN {X 0,Y 432.33,Z 372.63,A -85,B 0,C 180,E1 -9487.198,E2 -9487.198} C_VEL
LIN {X 0,Y 432.338,Z 372.628,A -85,B 0,C 180,E1 -9490.18,E2 -9490.18} C_VEL
LIN {X 0,Y 432.32,Z 372.631,A -85,B 0,C 180,E1 -9493.059,E2 -9493.059} C_VEL
LIN {X 0,Y 432.374,Z 372.628,A -85,B 0,C 180,E1 -9495.658,E2 -9495.658} C_VEL
LIN {X 0,Y 432.369,Z 372.623,A -85,B 0,C 180,E1 -9498.391,E2 -9498.391} C_VEL
LIN {X 0,Y 432.347,Z 372.629,A -85,B 0,C 180,E1 -9501.851,E2 -9501.851} C_VEL
LIN {X 0,Y 432.335,Z 372.634,A -85,B 0,C 180,E1 -9505.322,E2 -9505.322} C_VEL
LIN {X 0,Y 432.317,Z 372.63,A -85,B 0,C 180,E1 -9508.654,E2 -9508.654} C_VEL
LIN {X 0,Y 432.374,Z 372.63,A -85,B 0,C 180,E1 -9511.368,E2 -9511.368} C_VEL
LIN {X 0,Y 432.358,Z 372.625,A -85,B 0,C 180,E1 -9513.967,E2 -9513.967} C_VEL
LIN {X 0,Y 432.313,Z 372.635,A -85,B 0,C 180,E1 -9517.035,E2 -9517.035} C_VEL
LIN {X 0,Y 432.379,Z 372.622,A -85,B 0,C 180,E1 -9520.514,E2 -9520.514} C_VEL
LIN {X 0,Y 432.422,Z 372.617,A -85,B 0,C 180,E1 -9523.961,E2 -9523.961} C_VEL
LIN {X 0,Y 432.473,Z 372.611,A -85,B 0,C 180,E1 -9527.804,E2 -9527.804} C_VEL
LIN {X 0,Y 432.484,Z 372.61,A -85,B 0,C 180,E1 -9531.59,E2 -9531.59} C_VEL
LIN {X 0,Y 432.59,Z 372.597,A -85,B 0,C 180,E1 -9534.406,E2 -9534.406} C_VEL
LIN {X 0,Y 432.598,Z 372.595,A -85,B 0,C 180,E1 -9538.138,E2 -9538.138} C_VEL
LIN {X 0,Y 432.726,Z 372.578,A -85,B 0,C 180,E1 -9540,E2 -9540} C_VEL
LIN {X 0,Y 432.599,Z 372.601,A -85,B 0,C 180,E1 -9542.794,E2 -9542.794} C_VEL
LIN {X 0,Y 432.566,Z 372.602,A -85,B 0,C 180,E1 -9546.53,E2 -9546.53} C_VEL
LIN {X 0,Y 432.437,Z 372.616,A -85,B 0,C 180,E1 -9549.353,E2 -9549.353} C_VEL
LIN {X 0,Y 432.437,Z 372.622,A -85,B 0,C 180,E1 -9552.812,E2 -9552.812} C_VEL
LIN {X 0,Y 432.404,Z 372.623,A -85,B 0,C 180,E1 -9556.479,E2 -9556.479} C_VEL
LIN {X 0,Y 432.333,Z 372.628,A -85,B 0,C 180,E1 -9559.961,E2 -9559.961} C_VEL
LIN {X 0,Y 432.313,Z 372.633,A -85,B 0,C 180,E1 -9562.965,E2 -9562.965} C_VEL
LIN {X 0,Y 432.358,Z 372.626,A -85,B 0,C 180,E1 -9566.033,E2 -9566.033} C_VEL
LIN {X 0,Y 432.336,Z 372.628,A -85,B 0,C 180,E1 -9569.188,E2 -9569.188} C_VEL
LIN {X 0,Y 432.317,Z 372.636,A -85,B 0,C 180,E1 -9572.444,E2 -9572.444} C_VEL
LIN {X 0,Y 432.34,Z 372.627,A -85,B 0,C 180,E1 -9575.633,E2 -9575.633} C_VEL
LIN {X 0,Y 432.353,Z 372.629,A -85,B 0,C 180,E1 -9578.718,E2 -9578.718} C_VEL
LIN {X 0,Y 432.37,Z 372.624,A -85,B 0,C 180,E1 -9581.793,E2 -9581.793} C_VEL
LIN {X 0,Y 432.375,Z 372.63,A -85,B 0,C 180,E1 -9584.342,E2 -9584.342} C_VEL
LIN {X 0,Y 432.331,Z 372.634,A -85,B 0,C 180,E1 -9588.204,E2 -9588.204} C_VEL
LIN {X 0,Y 432.351,Z 372.625,A -85,B 0,C 180,E1 -9591.284,E2 -9591.284} C_VEL
LIN {X 0,Y 432.344,Z 372.631,A -85,B 0,C 180,E1 -9594.369,E2 -9594.369} C_VEL
LIN {X 0,Y 432.322,Z 372.63,A -85,B 0,C 180,E1 -9597.558,E2 -9597.558} C_VEL
LIN {X 0,Y 432.344,Z 372.627,A -85,B 0,C 180,E1 -9600.813,E2 -9600.813} C_VEL
LIN {X 0,Y 432.362,Z 372.63,A -85,B 0,C 180,E1 -9603.968,E2 -9603.968} C_VEL
LIN {X 0,Y 432.32,Z 372.634,A -85,B 0,C 180,E1 -9607.036,E2 -9607.036} C_VEL
LIN {X 0,Y 432.384,Z 372.764,A -85,B 0,C 180,E1 -9607.77,E2 -9607.77} C_VEL
LIN {X 0,Y 434.072,Z 382.078,A -85,B 0,C 180,E1 -9610.123,E2 -9610.123} C_VEL
LIN {X 0,Y 433.871,Z 388.53,A -85,B 0,C 180,E1 -9611.636,E2 -9611.636} C_VEL
LIN {X 0,Y 437.556,Z 406.874,A -85,B 0,C 180,E1 -9612.122,E2 -9612.122} C_VEL
LIN {X 0,Y 436.657,Z 495.743,A -85,B 0,C 180,E1 -9613.611,E2 -9613.611} C_VEL
LIN {X 0,Y 436.213,Z 509.582,A -85,B 0,C 180,E1 -9614.044,E2 -9614.044} C_VEL
LIN {X 0,Y 435.726,Z 521.968,A -85,B 0,C 180,E1 -9614.626,E2 -9614.626} C_VEL
LIN {X 0,Y 435.212,Z 533.808,A -85,B 0,C 180,E1 -9615.386,E2 -9615.386} C_VEL
LIN {X 0,Y 434.603,Z 545.117,A -85,B 0,C 180,E1 -9616.317,E2 -9616.317} C_VEL
LIN {X 0,Y 434.204,Z 551.427,A -85,B 0,C 180,E1 -9616.937,E2 -9616.937} C_VEL
LIN {X 0,Y 433.153,Z 556.02,A -85,B 0,C 180,E1 -9617.421,E2 -9617.421} C_VEL
LIN {X 0,Y 428.398,Z 565.852,A -85,B 0,C 180,E1 -9618.568,E2 -9618.568} C_VEL
LIN {X 0,Y 426.169,Z 570.998,A -85,B 0,C 180,E1 -9619.311,E2 -9619.311} C_VEL
LIN {X 0,Y 425.694,Z 573.405,A -85,B 0,C 180,E1 -9619.72,E2 -9619.72} C_VEL
LIN {X 0,Y 425.154,Z 580.894,A -85,B 0,C 180,E1 -9621.205,E2 -9621.205} C_VEL
LIN {X 0,Y 424.835,Z 585.726,A -85,B 0,C 180,E1 -9622.395,E2 -9622.395} C_VEL
LIN {X 0,Y 424.639,Z 590.417,A -85,B 0,C 180,E1 -9623.824,E2 -9623.824} C_VEL
LIN {X 0,Y 424.319,Z 594.015,A -85,B 0,C 180,E1 -9625.25,E2 -9625.25} C_VEL
LIN {X 0,Y 424.304,Z 595.869,A -85,B 0,C 180,E1 -9626.201,E2 -9626.201} C_VEL
LIN {X 0,Y 424.279,Z 597.266,A -85,B 0,C 180,E1 -9627.152,E2 -9627.152} C_VEL
LIN {X 0,Y 424.115,Z 598.876,A -85,B 0,C 180,E1 -9629.051,E2 -9629.051} C_VEL
LIN {X 0,Y 424.11,Z 599.11,A -85,B 0,C 180,E1 -9630,E2 -9630} C_VEL
LIN {X 0,Y 424.115,Z 598.923,A -85,B 0,C 180,E1 -9630.949,E2 -9630.949} C_VEL
LIN {X 0,Y 424.279,Z 597.373,A -85,B 0,C 180,E1 -9632.848,E2 -9632.848} C_VEL
LIN {X 0,Y 424.303,Z 596.022,A -85,B 0,C 180,E1 -9633.799,E2 -9633.799} C_VEL
LIN {X 0,Y 424.395,Z 593.166,A -85,B 0,C 180,E1 -9635.226,E2 -9635.226} C_VEL
LIN {X 0,Y 424.685,Z 588.777,A -85,B 0,C 180,E1 -9636.818,E2 -9636.818} C_VEL
LIN {X 0,Y 424.922,Z 584.287,A -85,B 0,C 180,E1 -9638.082,E2 -9638.082} C_VEL
LIN {X 0,Y 425.375,Z 577.987,A -85,B 0,C 180,E1 -9639.51,E2 -9639.51} C_VEL
LIN {X 0,Y 425.943,Z 570.099,A -85,B 0,C 180,E1 -9640.938,E2 -9640.938} C_VEL
LIN {X 0,Y 426.491,Z 562.057,A -85,B 0,C 180,E1 -9642.128,E2 -9642.128} C_VEL
LIN {X 0,Y 427.3,Z 552.234,A -85,B 0,C 180,E1 -9643.312,E2 -9643.312} C_VEL
LIN {X 0,Y 427.939,Z 541.193,A -85,B 0,C 180,E1 -9644.382,E2 -9644.382} C_VEL
LIN {X 0,Y 428.573,Z 530.361,A -85,B 0,C 180,E1 -9645.211,E2 -9645.211} C_VEL
LIN {X 0,Y 429.136,Z 518.396,A -85,B 0,C 180,E1 -9645.921,E2 -9645.921} C_VEL
LIN {X 0,Y 429.61,Z 506.136,A -85,B 0,C 180,E1 -9646.452,E2 -9646.452} C_VEL
LIN {X 0,Y 429.893,Z 493.53,A -85,B 0,C 180,E1 -9646.807,E2 -9646.807} C_VEL
LIN {X 0,Y 430.734,Z 407.095,A -85,B 0,C 180,E1 -9648.268,E2 -9648.268} C_VEL
LIN {X 0,Y 426.953,Z 388.849,A -85,B 0,C 180,E1 -9648.758,E2 -9648.758} C_VEL
LIN {X 0,Y 427.042,Z 382.528,A -85,B 0,C 180,E1 -9650.269,E2 -9650.269} C_VEL
LIN {X 0,Y 425.282,Z 373.518,A -85,B 0,C 180,E1 -9652.595,E2 -9652.595} C_VEL
LIN {X 0,Y 425.297,Z 373.51,A -85,B 0,C 180,E1 -9655.445,E2 -9655.445} C_VEL
LIN {X 0,Y 425.331,Z 373.501,A -85,B 0,C 180,E1 -9658.631,E2 -9658.631} C_VEL
LIN {X 0,Y 425.265,Z 373.516,A -85,B 0,C 180,E1 -9661.926,E2 -9661.926} C_VEL
LIN {X 0,Y 425.299,Z 373.505,A -85,B 0,C 180,E1 -9665.335,E2 -9665.335} C_VEL
LIN {X 0,Y 425.301,Z 373.504,A -85,B 0,C 180,E1 -9669.044,E2 -9669.044} C_VEL
LIN {X 0,Y 425.272,Z 373.507,A -85,B 0,C 180,E1 -9672.652,E2 -9672.652} C_VEL
LIN {X 0,Y 425.315,Z 373.505,A -85,B 0,C 180,E1 -9676.051,E2 -9676.051} C_VEL
LIN {X 0,Y 425.305,Z 373.503,A -85,B 0,C 180,E1 -9678.625,E2 -9678.625} C_VEL
LIN {X 0,Y 425.317,Z 373.503,A -85,B 0,C 180,E1 -9681.103,E2 -9681.103} C_VEL
LIN {X 0,Y 425.295,Z 373.504,A -85,B 0,C 180,E1 -9684.663,E2 -9684.663} C_VEL
LIN {X 0,Y 425.26,Z 373.51,A -85,B 0,C 180,E1 -9688.072,E2 -9688.072} C_VEL
LIN {X 0,Y 425.325,Z 373.506,A -85,B 0,C 180,E1 -9691.367,E2 -9691.367} C_VEL
LIN {X 0,Y 425.288,Z 373.505,A -85,B 0,C 180,E1 -9694.554,E2 -9694.554} C_VEL
LIN {X 0,Y 425.281,Z 373.51,A -85,B 0,C 180,E1 -9697.661,E2 -9697.661} C_VEL
LIN {X 0,Y 425.354,Z 373.498,A -85,B 0,C 180,E1 -9700.704,E2 -9700.704} C_VEL
LIN {X 0,Y 425.38,Z 373.497,A -85,B 0,C 180,E1 -9703.688,E2 -9703.688} C_VEL
LIN {X 0,Y 425.422,Z 373.492,A -85,B 0,C 180,E1 -9707.598,E2 -9707.598} C_VEL
LIN {X 0,Y 425.434,Z 373.491,A -85,B 0,C 180,E1 -9711.45,E2 -9711.45} C_VEL
LIN {X 0,Y 425.546,Z 373.473,A -85,B 0,C 180,E1 -9714.313,E2 -9714.313} C_VEL
LIN {X 0,Y 425.567,Z 373.47,A -85,B 0,C 180,E1 -9718.107,E2 -9718.107} C_VEL
LIN {X 0,Y 425.696,Z 373.454,A -85,B 0,C 180,E1 -9720,E2 -9720} C_VEL
LIN {X 0,Y 425.551,Z 373.477,A -85,B 0,C 180,E1 -9722.84,E2 -9722.84} C_VEL
LIN {X 0,Y 425.524,Z 373.479,A -85,B 0,C 180,E1 -9726.639,E2 -9726.639} C_VEL
LIN {X 0,Y 425.396,Z 373.493,A -85,B 0,C 180,E1 -9729.509,E2 -9729.509} C_VEL
LIN {X 0,Y 425.396,Z 373.499,A -85,B 0,C 180,E1 -9732.91,E2 -9732.91} C_VEL
LIN {X 0,Y 425.353,Z 373.501,A -85,B 0,C 180,E1 -9736.605,E2 -9736.605} C_VEL
LIN {X 0,Y 425.321,Z 373.501,A -85,B 0,C 180,E1 -9739.636,E2 -9739.636} C_VEL
LIN {X 0,Y 425.3,Z 373.505,A -85,B 0,C 180,E1 -9743.366,E2 -9743.366} C_VEL
LIN {X 0,Y 425.344,Z 373.504,A -85,B 0,C 180,E1 -9746.846,E2 -9746.846} C_VEL
LIN {X 0,Y 425.284,Z 373.505,A -85,B 0,C 180,E1 -9749.72,E2 -9749.72} C_VEL
LIN {X 0,Y 425.276,Z 373.509,A -85,B 0,C 180,E1 -9753.049,E2 -9753.049} C_VEL
LIN {X 0,Y 425.279,Z 373.507,A -85,B 0,C 180,E1 -9755.93,E2 -9755.93} C_VEL
LIN {X 0,Y 425.307,Z 373.505,A -85,B 0,C 180,E1 -9759.047,E2 -9759.047} C_VEL
LIN {X 0,Y 425.327,Z 373.506,A -85,B 0,C 180,E1 -9762.647,E2 -9762.647} C_VEL
LIN {X 0,Y 425.265,Z 373.511,A -85,B 0,C 180,E1 -9766.046,E2 -9766.046} C_VEL
LIN {X 0,Y 425.281,Z 373.506,A -85,B 0,C 180,E1 -9769.48,E2 -9769.48} C_VEL
LIN {X 0,Y 425.282,Z 373.512,A -85,B 0,C 180,E1 -9772.488,E2 -9772.488} C_VEL
LIN {X 0,Y 425.306,Z 373.505,A -85,B 0,C 180,E1 -9775.818,E2 -9775.818} C_VEL
LIN {X 0,Y 425.29,Z 373.506,A -85,B 0,C 180,E1 -9779.239,E2 -9779.239} C_VEL
LIN {X 0,Y 425.405,Z 373.655,A -85,B 0,C 180,E1 -9782.347,E2 -9782.347} C_VEL
LIN {X 0,Y 428.139,Z 387.244,A -85,B 0,C 180,E1 -9785.255,E2 -9785.255} C_VEL
LIN {X 0,Y 428.279,Z 392.451,A -85,B 0,C 180,E1 -9786.295,E2 -9786.295} C_VEL
LIN {X 0,Y 426.981,Z 411.841,A -85,B 0,C 180,E1 -9790.03,E2 -9790.03} C_VEL
LIN {X 0,Y 426.628,Z 418.322,A -85,B 0,C 180,E1 -9791.258,E2 -9791.258} C_VEL
LIN {X 0,Y 430.515,Z 444.014,A -85,B 0,C 180,E1 -9791.873,E2 -9791.873} C_VEL
LIN {X 0,Y 429.615,Z 526.592,A -85,B 0,C 180,E1 -9793.273,E2 -9793.273} C_VEL
LIN {X 0,Y 429.169,Z 539.844,A -85,B 0,C 180,E1 -9793.684,E2 -9793.684} C_VEL
LIN {X 0,Y 428.552,Z 551.999,A -85,B 0,C 180,E1 -9794.24,E2 -9794.24} C_VEL
LIN {X 0,Y 427.842,Z 564.27,A -85,B 0,C 180,E1 -9795.006,E2 -9795.006} C_VEL
LIN {X 0,Y 427.056,Z 575.499,A -85,B 0,C 180,E1 -9795.917,E2 -9795.917} C_VEL
LIN {X 0,Y 426.4,Z 586.327,A -85,B 0,C 180,E1 -9797.023,E2 -9797.023} C_VEL
LIN {X 0,Y 425.847,Z 594.877,A -85,B 0,C 180,E1 -9798.095,E2 -9798.095} C_VEL
LIN {X 0,Y 425.259,Z 602.765,A -85,B 0,C 180,E1 -9799.285,E2 -9799.285} C_VEL
LIN {X 0,Y 424.787,Z 610.475,A -85,B 0,C 180,E1 -9800.717,E2 -9800.717} C_VEL
LIN {X 0,Y 424.415,Z 617.586,A -85,B 0,C 180,E1 -9802.388,E2 -9802.388} C_VEL
LIN {X 0,Y 424.217,Z 622.062,A -85,B 0,C 180,E1 -9803.733,E2 -9803.733} C_VEL
LIN {X 0,Y 424.2,Z 625.94,A -85,B 0,C 180,E1 -9805.248,E2 -9805.248} C_VEL
LIN {X 0,Y 424.101,Z 627.804,A -85,B 0,C 180,E1 -9806.199,E2 -9806.199} C_VEL
LIN {X 0,Y 424.134,Z 629.206,A -85,B 0,C 180,E1 -9807.151,E2 -9807.151} C_VEL
LIN {X 0,Y 424.143,Z 630.205,A -85,B 0,C 180,E1 -9808.101,E2 -9808.101} C_VEL
LIN {X 0,Y 424.111,Z 630.814,A -85,B 0,C 180,E1 -9809.051,E2 -9809.051} C_VEL
LIN {X 0,Y 424.108,Z 631.03,A -85,B 0,C 180,E1 -9810,E2 -9810} C_VEL
LIN {X 0,Y 424.143,Z 630.204,A -85,B 0,C 180,E1 -9811.899,E2 -9811.899} C_VEL
LIN {X 0,Y 424.134,Z 629.205,A -85,B 0,C 180,E1 -9812.849,E2 -9812.849} C_VEL
LIN {X 0,Y 424.101,Z 627.802,A -85,B 0,C 180,E1 -9813.801,E2 -9813.801} C_VEL
LIN {X 0,Y 424.207,Z 624.858,A -85,B 0,C 180,E1 -9815.228,E2 -9815.228} C_VEL
LIN {X 0,Y 424.299,Z 620.871,A -85,B 0,C 180,E1 -9816.658,E2 -9816.658} C_VEL
LIN {X 0,Y 424.546,Z 614.744,A -85,B 0,C 180,E1 -9818.328,E2 -9818.328} C_VEL
LIN {X 0,Y 424.926,Z 608.052,A -85,B 0,C 180,E1 -9819.76,E2 -9819.76} C_VEL
LIN {X 0,Y 425.458,Z 599.753,A -85,B 0,C 180,E1 -9821.192,E2 -9821.192} C_VEL
LIN {X 0,Y 426.094,Z 591.252,A -85,B 0,C 180,E1 -9822.381,E2 -9822.381} C_VEL
LIN {X 0,Y 426.718,Z 581.519,A -85,B 0,C 180,E1 -9823.494,E2 -9823.494} C_VEL
LIN {X 0,Y 427.427,Z 570.357,A -85,B 0,C 180,E1 -9824.521,E2 -9824.521} C_VEL
LIN {X 0,Y 428.13,Z 558.971,A -85,B 0,C 180,E1 -9825.349,E2 -9825.349} C_VEL
LIN {X 0,Y 428.777,Z 547.289,A -85,B 0,C 180,E1 -9825.996,E2 -9825.996} C_VEL
LIN {X 0,Y 429.34,Z 534.745,A -85,B 0,C 180,E1 -9826.493,E2 -9826.493} C_VEL
LIN {X 0,Y 429.686,Z 522.03,A -85,B 0,C 180,E1 -9826.816,E2 -9826.816} C_VEL
LIN {X 0,Y 430.391,Z 442.451,A -85,B 0,C 180,E1 -9828.154,E2 -9828.154} C_VEL
LIN {X 0,Y 426.601,Z 418.189,A -85,B 0,C 180,E1 -9828.744,E2 -9828.744} C_VEL
LIN {X 0,Y 427.709,Z 400.181,A -85,B 0,C 180,E1 -9832.205,E2 -9832.205} C_VEL
LIN {X 0,Y 428.345,Z 388.521,A -85,B 0,C 180,E1 -9834.474,E2 -9834.474} C_VEL
LIN {X 0,Y 425.855,Z 375.703,A -85,B 0,C 180,E1 -9837.196,E2 -9837.196} C_VEL
LIN {X 0,Y 425.376,Z 373.499,A -85,B 0,C 180,E1 -9837.689,E2 -9837.689} C_VEL
LIN {X 0,Y 425.287,Z 373.51,A -85,B 0,C 180,E1 -9840.815,E2 -9840.815} C_VEL
LIN {X 0,Y 425.31,Z 373.504,A -85,B 0,C 180,E1 -9844.287,E2 -9844.287} C_VEL
LIN {X 0,Y 425.284,Z 373.513,A -85,B 0,C 180,E1 -9847.693,E2 -9847.693} C_VEL
LIN {X 0,Y 425.281,Z 373.506,A -85,B 0,C 180,E1 -9850.52,E2 -9850.52} C_VEL
LIN {X 0,Y 425.265,Z 373.511,A -85,B 0,C 180,E1 -9853.954,E2 -9853.954} C_VEL
LIN {X 0,Y 425.327,Z 373.506,A -85,B 0,C 180,E1 -9857.353,E2 -9857.353} C_VEL
LIN {X 0,Y 425.318,Z 373.504,A -85,B 0,C 180,E1 -9861.103,E2 -9861.103} C_VEL
LIN {X 0,Y 425.295,Z 373.505,A -85,B 0,C 180,E1 -9864.664,E2 -9864.664} C_VEL
LIN {X 0,Y 425.26,Z 373.509,A -85,B 0,C 180,E1 -9868.073,E2 -9868.073} C_VEL
LIN {X 0,Y 425.331,Z 373.507,A -85,B 0,C 180,E1 -9871.368,E2 -9871.368} C_VEL
LIN {X 0,Y 425.288,Z 373.506,A -85,B 0,C 180,E1 -9874.554,E2 -9874.554} C_VEL
LIN {X 0,Y 425.281,Z 373.509,A -85,B 0,C 180,E1 -9877.661,E2 -9877.661} C_VEL
LIN {X 0,Y 425.354,Z 373.499,A -85,B 0,C 180,E1 -9880.704,E2 -9880.704} C_VEL
LIN {X 0,Y 425.38,Z 373.495,A -85,B 0,C 180,E1 -9883.688,E2 -9883.688} C_VEL
LIN {X 0,Y 425.422,Z 373.49,A -85,B 0,C 180,E1 -9887.598,E2 -9887.598} C_VEL
LIN {X 0,Y 425.434,Z 373.49,A -85,B 0,C 180,E1 -9891.45,E2 -9891.45} C_VEL
LIN {X 0,Y 425.546,Z 373.474,A -85,B 0,C 180,E1 -9894.313,E2 -9894.313} C_VEL
LIN {X 0,Y 425.568,Z 373.47,A -85,B 0,C 180,E1 -9898.107,E2 -9898.107} C_VEL
LIN {X 0,Y 425.696,Z 373.454,A -85,B 0,C 180,E1 -9900,E2 -9900} C_VEL
LIN {X 0,Y 425.551,Z 373.479,A -85,B 0,C 180,E1 -9902.84,E2 -9902.84} C_VEL
LIN {X 0,Y 425.523,Z 373.48,A -85,B 0,C 180,E1 -9906.656,E2 -9906.656} C_VEL
LIN {X 0,Y 425.396,Z 373.492,A -85,B 0,C 180,E1 -9909.51,E2 -9909.51} C_VEL
LIN {X 0,Y 425.396,Z 373.497,A -85,B 0,C 180,E1 -9912.91,E2 -9912.91} C_VEL
LIN {X 0,Y 425.353,Z 373.503,A -85,B 0,C 180,E1 -9916.605,E2 -9916.605} C_VEL
LIN {X 0,Y 425.321,Z 373.501,A -85,B 0,C 180,E1 -9919.636,E2 -9919.636} C_VEL
LIN {X 0,Y 425.301,Z 373.504,A -85,B 0,C 180,E1 -9923.366,E2 -9923.366} C_VEL
LIN {X 0,Y 425.342,Z 373.502,A -85,B 0,C 180,E1 -9926.845,E2 -9926.845} C_VEL
LIN {X 0,Y 425.284,Z 373.506,A -85,B 0,C 180,E1 -9929.72,E2 -9929.72} C_VEL
LIN {X 0,Y 425.276,Z 373.508,A -85,B 0,C 180,E1 -9933.049,E2 -9933.049} C_VEL
LIN {X 0,Y 425.279,Z 373.508,A -85,B 0,C 180,E1 -9935.93,E2 -9935.93} C_VEL
LIN {X 0,Y 425.306,Z 373.504,A -85,B 0,C 180,E1 -9939.046,E2 -9939.046} C_VEL
LIN {X 0,Y 425.328,Z 373.504,A -85,B 0,C 180,E1 -9942.647,E2 -9942.647} C_VEL
LIN {X 0,Y 425.291,Z 373.505,A -85,B 0,C 180,E1 -9945.283,E2 -9945.283} C_VEL
LIN {X 0,Y 425.272,Z 373.51,A -85,B 0,C 180,E1 -9948.622,E2 -9948.622} C_VEL
LIN {X 0,Y 425.313,Z 373.502,A -85,B 0,C 180,E1 -9951.104,E2 -9951.104} C_VEL
LIN {X 0,Y 425.299,Z 373.506,A -85,B 0,C 180,E1 -9954.665,E2 -9954.665} C_VEL
LIN {X 0,Y 425.265,Z 373.515,A -85,B 0,C 180,E1 -9958.074,E2 -9958.074} C_VEL
LIN {X 0,Y 425.332,Z 373.5,A -85,B 0,C 180,E1 -9961.369,E2 -9961.369} C_VEL
LIN {X 0,Y 425.355,Z 373.498,A -85,B 0,C 180,E1 -9963.506,E2 -9963.506} C_VEL
LIN {X 0,Y 425.307,Z 373.51,A -85,B 0,C 180,E1 -9966.635,E2 -9966.635} C_VEL
LIN {X 0,Y 425.302,Z 373.619,A -85,B 0,C 180,E1 -9967.535,E2 -9967.535} C_VEL
LIN {X 0,Y 427.132,Z 383.361,A -85,B 0,C 180,E1 -9970.037,E2 -9970.037} C_VEL
LIN {X 0,Y 426.956,Z 388.818,A -85,B 0,C 180,E1 -9971.334,E2 -9971.334} C_VEL
LIN {X 0,Y 430.82,Z 407.579,A -85,B 0,C 180,E1 -9971.84,E2 -9971.84} C_VEL
LIN {X 0,Y 429.882,Z 496.026,A -85,B 0,C 180,E1 -9973.345,E2 -9973.345} C_VEL
LIN {X 0,Y 429.409,Z 509.86,A -85,B 0,C 180,E1 -9973.785,E2 -9973.785} C_VEL
LIN {X 0,Y 428.893,Z 522.242,A -85,B 0,C 180,E1 -9974.375,E2 -9974.375} C_VEL
LIN {X 0,Y 428.357,Z 534.081,A -85,B 0,C 180,E1 -9975.147,E2 -9975.147} C_VEL
LIN {X 0,Y 427.69,Z 545.799,A -85,B 0,C 180,E1 -9976.13,E2 -9976.13} C_VEL
LIN {X 0,Y 427.002,Z 555.652,A -85,B 0,C 180,E1 -9977.162,E2 -9977.162} C_VEL
LIN {X 0,Y 426.339,Z 564.825,A -85,B 0,C 180,E1 -9978.35,E2 -9978.35} C_VEL
LIN {X 0,Y 425.694,Z 573.405,A -85,B 0,C 180,E1 -9979.72,E2 -9979.72} C_VEL
LIN {X 0,Y 424.772,Z 576.921,A -85,B 0,C 180,E1 -9980.35,E2 -9980.35} C_VEL
LIN {X 0,Y 421.511,Z 582.274,A -85,B 0,C 180,E1 -9981.395,E2 -9981.395} C_VEL
LIN {X 0,Y 418.352,Z 586.912,A -85,B 0,C 180,E1 -9982.512,E2 -9982.512} C_VEL
LIN {X 0,Y 417.601,Z 589.304,A -85,B 0,C 180,E1 -9983.245,E2 -9983.245} C_VEL
LIN {X 0,Y 417.349,Z 593.221,A -85,B 0,C 180,E1 -9984.686,E2 -9984.686} C_VEL
LIN {X 0,Y 417.213,Z 596.137,A -85,B 0,C 180,E1 -9986.137,E2 -9986.137} C_VEL
LIN {X 0,Y 417.214,Z 597.533,A -85,B 0,C 180,E1 -9987.103,E2 -9987.103} C_VEL
LIN {X 0,Y 417.036,Z 599.143,A -85,B 0,C 180,E1 -9989.034,E2 -9989.034} C_VEL
LIN {X 0,Y 417.028,Z 599.377,A -85,B 0,C 180,E1 -9990,E2 -9990} C_VEL
LIN {X 0,Y 417.036,Z 599.189,A -85,B 0,C 180,E1 -9990.966,E2 -9990.966} C_VEL
LIN {X 0,Y 417.214,Z 597.639,A -85,B 0,C 180,E1 -9992.897,E2 -9992.897} C_VEL
LIN {X 0,Y 417.212,Z 596.289,A -85,B 0,C 180,E1 -9993.863,E2 -9993.863} C_VEL
LIN {X 0,Y 417.346,Z 593.431,A -85,B 0,C 180,E1 -9995.314,E2 -9995.314} C_VEL
LIN {X 0,Y 417.606,Z 589.406,A -85,B 0,C 180,E1 -9996.816,E2 -9996.816} C_VEL
LIN {X 0,Y 417.891,Z 584.552,A -85,B 0,C 180,E1 -9998.218,E2 -9998.218} C_VEL
LIN {X 0,Y 418.381,Z 578.252,A -85,B 0,C 180,E1 -9999.67,E2 -9999.67} C_VEL
LIN {X 0,Y 418.989,Z 570.363,A -85,B 0,C 180,E1 -10001.122,E2 -10001.122} C_VEL
LIN {X 0,Y 419.563,Z 562.32,A -85,B 0,C 180,E1 -10002.331,E2 -10002.331} C_VEL
LIN {X 0,Y 420.402,Z 552.497,A -85,B 0,C 180,E1 -10003.535,E2 -10003.535} C_VEL
LIN {X 0,Y 421.067,Z 541.455,A -85,B 0,C 180,E1 -10004.622,E2 -10004.622} C_VEL
LIN {X 0,Y 421.726,Z 530.622,A -85,B 0,C 180,E1 -10005.464,E2 -10005.464} C_VEL
LIN {X 0,Y 422.341,Z 518.654,A -85,B 0,C 180,E1 -10006.184,E2 -10006.184} C_VEL
LIN {X 0,Y 422.816,Z 506.391,A -85,B 0,C 180,E1 -10006.724,E2 -10006.724} C_VEL
LIN {X 0,Y 423.114,Z 493.774,A -85,B 0,C 180,E1 -10007.085,E2 -10007.085} C_VEL
LIN {X 0,Y 424.003,Z 407.97,A -85,B 0,C 180,E1 -10008.557,E2 -10008.557} C_VEL
LIN {X 0,Y 420.048,Z 389.1,A -85,B 0,C 180,E1 -10009.081,E2 -10009.081} C_VEL
LIN {X 0,Y 420.227,Z 385.315,A -85,B 0,C 180,E1 -10009.987,E2 -10009.987} C_VEL
LIN {X 0,Y 418.463,Z 375.544,A -85,B 0,C 180,E1 -10012.524,E2 -10012.524} C_VEL
LIN {X 0,Y 418.244,Z 374.394,A -85,B 0,C 180,E1 -10012.866,E2 -10012.866} C_VEL
LIN {X 0,Y 418.272,Z 374.386,A -85,B 0,C 180,E1 -10015.903,E2 -10015.903} C_VEL
LIN {X 0,Y 418.265,Z 374.38,A -85,B 0,C 180,E1 -10019.161,E2 -10019.161} C_VEL
LIN {X 0,Y 418.257,Z 374.381,A -85,B 0,C 180,E1 -10022.843,E2 -10022.843} C_VEL
LIN {X 0,Y 418.247,Z 374.385,A -85,B 0,C 180,E1 -10026.238,E2 -10026.238} C_VEL
LIN {X 0,Y 418.253,Z 374.387,A -85,B 0,C 180,E1 -10029.681,E2 -10029.681} C_VEL
LIN {X 0,Y 418.227,Z 374.386,A -85,B 0,C 180,E1 -10032.32,E2 -10032.32} C_VEL
LIN {X 0,Y 418.256,Z 374.382,A -85,B 0,C 180,E1 -10035.111,E2 -10035.111} C_VEL
LIN {X 0,Y 418.289,Z 374.384,A -85,B 0,C 180,E1 -10037.773,E2 -10037.773} C_VEL
LIN {X 0,Y 418.26,Z 374.387,A -85,B 0,C 180,E1 -10041.559,E2 -10041.559} C_VEL
LIN {X 0,Y 418.254,Z 374.384,A -85,B 0,C 180,E1 -10045.158,E2 -10045.158} C_VEL
LIN {X 0,Y 418.24,Z 374.389,A -85,B 0,C 180,E1 -10047.471,E2 -10047.471} C_VEL
LIN {X 0,Y 418.262,Z 374.381,A -85,B 0,C 180,E1 -10050.895,E2 -10050.895} C_VEL
LIN {X 0,Y 418.264,Z 374.381,A -85,B 0,C 180,E1 -10054.095,E2 -10054.095} C_VEL
LIN {X 0,Y 418.231,Z 374.389,A -85,B 0,C 180,E1 -10057.263,E2 -10057.263} C_VEL
LIN {X 0,Y 418.276,Z 374.379,A -85,B 0,C 180,E1 -10060.364,E2 -10060.364} C_VEL
LIN {X 0,Y 418.309,Z 374.381,A -85,B 0,C 180,E1 -10063.404,E2 -10063.404} C_VEL
LIN {X 0,Y 418.347,Z 374.373,A -85,B 0,C 180,E1 -10066.993,E2 -10066.993} C_VEL
LIN {X 0,Y 418.352,Z 374.369,A -85,B 0,C 180,E1 -10070.329,E2 -10070.329} C_VEL
LIN {X 0,Y 418.485,Z 374.359,A -85,B 0,C 180,E1 -10073.249,E2 -10073.249} C_VEL
LIN {X 0,Y 418.335,Z 374.379,A -85,B 0,C 180,E1 -10075.181,E2 -10075.181} C_VEL
LIN {X 0,Y 418.537,Z 374.346,A -85,B 0,C 180,E1 -10078.075,E2 -10078.075} C_VEL
LIN {X 0,Y 418.666,Z 374.33,A -85,B 0,C 180,E1 -10080,E2 -10080} C_VEL
LIN {X 0,Y 418.505,Z 374.355,A -85,B 0,C 180,E1 -10082.888,E2 -10082.888} C_VEL
LIN {X 0,Y 418.486,Z 374.357,A -85,B 0,C 180,E1 -10086.751,E2 -10086.751} C_VEL
LIN {X 0,Y 418.353,Z 374.37,A -85,B 0,C 180,E1 -10089.671,E2 -10089.671} C_VEL
LIN {X 0,Y 418.347,Z 374.376,A -85,B 0,C 180,E1 -10093.006,E2 -10093.006} C_VEL
LIN {X 0,Y 418.305,Z 374.381,A -85,B 0,C 180,E1 -10096.736,E2 -10096.736} C_VEL
LIN {X 0,Y 418.264,Z 374.38,A -85,B 0,C 180,E1 -10099.791,E2 -10099.791} C_VEL
LIN {X 0,Y 418.231,Z 374.391,A -85,B 0,C 180,E1 -10102.737,E2 -10102.737} C_VEL
LIN {X 0,Y 418.264,Z 374.38,A -85,B 0,C 180,E1 -10105.905,E2 -10105.905} C_VEL
LIN {X 0,Y 418.258,Z 374.383,A -85,B 0,C 180,E1 -10109.163,E2 -10109.163} C_VEL
LIN {X 0,Y 418.251,Z 374.386,A -85,B 0,C 180,E1 -10112.845,E2 -10112.845} C_VEL
LIN {X 0,Y 418.243,Z 374.386,A -85,B 0,C 180,E1 -10116.239,E2 -10116.239} C_VEL
LIN {X 0,Y 418.261,Z 374.381,A -85,B 0,C 180,E1 -10119.681,E2 -10119.681} C_VEL
LIN {X 0,Y 418.281,Z 374.383,A -85,B 0,C 180,E1 -10122.33,E2 -10122.33} C_VEL
LIN {X 0,Y 418.251,Z 374.383,A -85,B 0,C 180,E1 -10125.112,E2 -10125.112} C_VEL
LIN {X 0,Y 418.239,Z 374.384,A -85,B 0,C 180,E1 -10127.768,E2 -10127.768} C_VEL
LIN {X 0,Y 418.257,Z 374.385,A -85,B 0,C 180,E1 -10130.619,E2 -10130.619} C_VEL
LIN {X 0,Y 418.244,Z 374.386,A -85,B 0,C 180,E1 -10133.977,E2 -10133.977} C_VEL
LIN {X 0,Y 418.259,Z 374.381,A -85,B 0,C 180,E1 -10137.156,E2 -10137.156} C_VEL
LIN {X 0,Y 418.268,Z 374.383,A -85,B 0,C 180,E1 -10140.896,E2 -10140.896} C_VEL
LIN {X 0,Y 418.348,Z 374.456,A -85,B 0,C 180,E1 -10142.057,E2 -10142.057} C_VEL
LIN {X 0,Y 420.957,Z 387.302,A -85,B 0,C 180,E1 -10144.867,E2 -10144.867} C_VEL
LIN {X 0,Y 421.446,Z 392.21,A -85,B 0,C 180,E1 -10145.886,E2 -10145.886} C_VEL
LIN {X 0,Y 420.059,Z 411.53,A -85,B 0,C 180,E1 -10149.676,E2 -10149.676} C_VEL
LIN {X 0,Y 419.717,Z 417.895,A -85,B 0,C 180,E1 -10150.927,E2 -10150.927} C_VEL
LIN {X 0,Y 423.745,Z 443.921,A -85,B 0,C 180,E1 -10151.576,E2 -10151.576} C_VEL
LIN {X 0,Y 422.835,Z 526.338,A -85,B 0,C 180,E1 -10152.997,E2 -10152.997} C_VEL
LIN {X 0,Y 422.345,Z 539.585,A -85,B 0,C 180,E1 -10153.412,E2 -10153.412} C_VEL
LIN {X 0,Y 421.724,Z 551.738,A -85,B 0,C 180,E1 -10153.978,E2 -10153.978} C_VEL
LIN {X 0,Y 420.952,Z 564.005,A -85,B 0,C 180,E1 -10154.755,E2 -10154.755} C_VEL
LIN {X 0,Y 420.133,Z 575.504,A -85,B 0,C 180,E1 -10155.706,E2 -10155.706} C_VEL
LIN {X 0,Y 419.446,Z 586.061,A -85,B 0,C 180,E1 -10156.804,E2 -10156.804} C_VEL
LIN {X 0,Y 418.866,Z 594.611,A -85,B 0,C 180,E1 -10157.894,E2 -10157.894} C_VEL
LIN {X 0,Y 418.261,Z 602.499,A -85,B 0,C 180,E1 -10159.104,E2 -10159.104} C_VEL
LIN {X 0,Y 417.751,Z 610.208,A -85,B 0,C 180,E1 -10160.559,E2 -10160.559} C_VEL
LIN {X 0,Y 417.354,Z 617.319,A -85,B 0,C 180,E1 -10162.258,E2 -10162.258} C_VEL
LIN {X 0,Y 417.124,Z 622.194,A -85,B 0,C 180,E1 -10163.761,E2 -10163.761} C_VEL
LIN {X 0,Y 417.107,Z 625.673,A -85,B 0,C 180,E1 -10165.167,E2 -10165.167} C_VEL
LIN {X 0,Y 417.016,Z 627.537,A -85,B 0,C 180,E1 -10166.135,E2 -10166.135} C_VEL
LIN {X 0,Y 417.032,Z 628.939,A -85,B 0,C 180,E1 -10167.102,E2 -10167.102} C_VEL
LIN {X 0,Y 417.069,Z 629.939,A -85,B 0,C 180,E1 -10168.069,E2 -10168.069} C_VEL
LIN {X 0,Y 417.032,Z 630.548,A -85,B 0,C 180,E1 -10169.034,E2 -10169.034} C_VEL
LIN {X 0,Y 417.027,Z 630.764,A -85,B 0,C 180,E1 -10170,E2 -10170} C_VEL
LIN {X 0,Y 417.069,Z 629.938,A -85,B 0,C 180,E1 -10171.931,E2 -10171.931} C_VEL
LIN {X 0,Y 417.032,Z 628.937,A -85,B 0,C 180,E1 -10172.898,E2 -10172.898} C_VEL
